Yaskawa INFORM job: X2_38-47,64(1)(90,180)_HARDOX.JBI

/JOB
//NAME X2_38-47,64(1)(90,180)_HARDOX
//POS
///NPOS 504,504,504,30,0,0
///TOOL 0
///POSTYPE PULSE
///PULSE
C00000=-10776,-116726,-133110,1428,79202,268
C00001=-121301,-101656,-130574,-15140,106953,-26685
C00002=-120740,-100574,-124017,-14929,103680,-26084
C00003=-120691,-100743,-123189,-14892,103111,-25997
C00004=-120691,-101012,-123023,-14875,102879,-25968
C00005=-120694,-100727,-123199,-14892,103125,-25999
C00006=-120263,-93974,-120700,-15099,105066,-26103
C00007=-120694,-100727,-123199,-14892,103125,-25999
C00008=-121303,-103883,-129892,-15002,105440,-26491
C00009=-121309,-101301,-130428,-15148,107041,-26699
C00010=-120755,-99767,-124232,-14968,104207,-26155
C00011=-120700,-99774,-123449,-14938,103747,-26079
C00012=-120700,-100712,-122892,-14879,102948,-25979
C00013=-120685,-100384,-123078,-14901,103225,-26009
C00014=-120255,-93653,-120581,-15108,105156,-26112
C00015=-120685,-100384,-123078,-14901,103225,-26009
C00016=-121293,-103472,-129753,-15014,105563,-26504
C00017=-114791,-117911,-130965,-19588,74628,-29967
C00018=-114769,-122713,-124135,-20312,68344,-28880
C00019=-114477,-110584,-116158,-20272,69659,-29005
C00020=-114421,-108517,-114081,-20323,69469,-28951
C00021=-114421,-108669,-113508,-20377,69064,-28879
C00022=-114502,-108614,-114130,-20291,69431,-28974
C00023=-116741,-105993,-113204,-19215,69642,-29832
C00024=-114502,-108614,-114130,-20291,69431,-28974
C00025=-119599,-132627,-121815,-19129,61042,-29452
C00026=-135151,-106131,-113172,-10502,66286,-36044
C00027=-134382,-104032,-112419,-10838,66989,-35834
C00028=-133562,-101757,-111587,-11194,67742,-35614
C00029=-135151,-106131,-113172,-10502,66286,-36044
C00030=-114538,-130880,-126635,-20790,65904,-28347
C00031=-100256,-119338,-132400,-19781,92736,17009
C00032=-115252,-134637,-128783,-15911,82002,19716
C00033=-118597,-124593,-122817,-15129,82811,18454
C00034=-119849,-120977,-120499,-14834,83003,18000
C00035=-119848,-121103,-118880,-14863,81976,18124
C00036=-119849,-120977,-120499,-14834,83003,18000
C00037=-134184,-142802,-124917,-2858,68148,11180
C00038=-133176,-135816,-122960,-3144,70568,11480
C00039=-134184,-142802,-124917,-2858,68148,11180
C00040=-110326,-92448,-108322,-23569,98205,21456
C00041=-112623,-92143,-108201,-23254,97666,20755
C00042=-110326,-92448,-108322,-23569,98205,21456
C00043=-105090,-96290,-113946,-24376,100996,22735
C00044=-105112,-88407,-119445,-25319,107768,21250
C00045=-126458,-130213,-127441,18734,86324,-24062
C00046=-122565,-122494,-122126,18005,86127,-22734
C00047=-121090,-119592,-120022,17718,85999,-22241
C00048=-121089,-119765,-118419,17734,84972,-22390
C00049=-121090,-119592,-120022,17718,85999,-22241
C00050=-121090,-119716,-118696,17731,85160,-22363
C00051=-120619,-113401,-116618,17615,86937,-21943
C00052=-121090,-119716,-118696,17731,85160,-22363
C00053=-120691,-116357,-117549,17638,86049,-22096
C00054=-118089,-117386,-117887,17123,85200,-21315
C00055=-120691,-116357,-117549,17638,86049,-22096
C00056=-125936,-126318,-124843,18636,86589,-23840
C00057=-125953,-122568,-132013,18690,92614,-22924
C00058=-117644,-124381,-130105,-6983,115370,67992
C00059=-119593,-136528,-130318,-6950,109138,67660
C00060=-120425,-140611,-129416,-6959,106433,67520
C00061=-120425,-140322,-128375,-6938,105944,67549
C00062=-120287,-139878,-129033,-6943,106584,67561
C00063=-121808,-147552,-131144,-7070,103828,67181
C00064=-120287,-139878,-129033,-6943,106584,67561
C00065=-117523,-124132,-129146,-6933,114921,68065
C00066=-117634,-108923,-132591,-7489,118176,67765
C00067=-119077,-97405,-129626,-2848,111310,9091
C00068=-112934,-122170,-124968,-9693,82630,11419
C00069=-114889,-112052,-118675,-9157,83718,10686
C00070=-115614,-108714,-115508,-8968,83408,10468
C00071=-115614,-108962,-114752,-8976,82823,10510
C00072=-115614,-108688,-115602,-8966,83479,10463
C00073=-130338,-117040,-117457,5173,77211,4432
C00074=-129550,-114521,-116623,4914,77941,4728
C00075=-131152,-119600,-118288,5441,76463,4123
C00076=-115450,-106601,-114144,-9007,83670,10503
C00077=-117654,-103921,-113183,-8408,84218,9737
C00078=-115450,-106601,-114144,-9007,83670,10503
C00079=-112794,-119726,-122752,-9732,82540,11472
C00080=-112816,-114614,-129461,-9677,89201,10949
C00081=-124267,-125778,-125536,12618,81617,-14637
C00082=-121749,-115664,-119377,11934,82621,-13684
C00083=-120813,-112238,-116231,11692,82317,-13397
C00084=-120812,-112414,-115451,11705,81758,-13450
C00085=-120848,-112349,-116241,11703,82272,-13413
C00086=-119586,-107060,-114409,11339,83657,-12862
C00087=-120848,-112349,-116241,11703,82272,-13413
C00088=-124307,-126037,-124767,12644,81031,-14711
C00089=-124281,-122814,-131176,12539,86499,-14147
C00090=-130647,-155525,-127944,40400,54320,-55258
C00091=-124412,-146323,-123540,36852,53123,-52512
C00092=-122059,-142698,-121760,35413,52755,-51453
C00093=-119008,-142706,-121763,33902,51510,-50382
C00094=-122059,-142698,-121760,35413,52755,-51453
C00095=-119813,-142714,-121776,34308,51836,-50667
C00096=-119829,-137326,-119074,33845,52767,-50322
C00097=-119813,-142714,-121776,34308,51836,-50667
C00098=-119893,-119020,-120433,30427,61542,-47434
C00099=-120958,-113296,-116932,30756,62602,-47571
C00100=-120971,-118070,-117370,31352,60722,-48150
C00101=-120958,-113296,-116932,30756,62602,-47571
C00102=-130647,-155525,-127944,40400,54320,-55258
C00103=-121972,-140000,-127461,3525,22047,-40740
C00104=-114503,-126631,-127045,-28228,88345,-28238
C00105=-115418,-120062,-121213,-28067,87856,-28460
C00106=-115767,-117777,-118144,-28010,87108,-28410
C00107=-115767,-117863,-117333,-28016,86625,-28294
C00108=-115798,-117876,-117463,-28010,86680,-28319
C00109=-115506,-111666,-115391,-28051,88476,-28642
C00110=-115798,-117876,-117463,-28010,86680,-28319
C00111=-114535,-126949,-125608,-28226,87406,-28022
C00112=-81132,-132100,-132064,-22325,96940,-18748
C00113=-82014,-125321,-126186,-22252,96583,-18997
C00114=-82351,-123063,-123074,-22185,95795,-18971
C00115=-82354,-123167,-122323,-22159,95314,-18883
C00116=-82329,-123147,-122467,-22165,95412,-18892
C00117=-83163,-116500,-120334,-22218,97147,-19515
C00118=-82329,-123147,-122467,-22165,95412,-18892
C00119=-81992,-125617,-124767,-22197,95637,-18813
C00120=-81110,-132470,-130662,-22266,95968,-18558
C00121=-88413,-113418,-132573,-32131,117765,-52556
C00122=-88284,-148255,-125485,-32887,110398,-70729
C00123=-90408,-157751,-124889,-32381,105124,-70012
C00124=-91344,-160468,-123864,-32301,103041,-69779
C00125=-91347,-158891,-122215,-32272,102866,-69728
C00126=-106792,-136481,-118062,-29763,111204,-74713
C00127=-106248,-142899,-119829,-29161,109458,-74003
C00128=-106792,-136481,-118062,-29763,111204,-74713
C00129=-72811,-175927,-123443,-35029,98716,-64074
C00130=-76149,-179694,-124176,-35896,96158,-64586
C00131=-72811,-175927,-123443,-35029,98716,-64074
C00132=-69241,-166504,-125806,-34856,105362,-64752
C00133=-100814,-129767,-126176,-13403,120642,-68982
C00134=-124653,-147507,-132240,11278,113041,-68250
C00135=-122082,-159833,-132453,11465,106593,-67927
C00136=-120959,-163108,-131284,11603,104077,-67764
C00137=-120958,-161905,-130051,11594,103939,-67777
C00138=-120958,-161991,-130311,11601,104052,-67766
C00139=-120981,-170969,-132443,11421,100817,-68083
C00140=-120958,-161991,-130311,11601,104052,-67766
C00141=-120973,-170778,-133362,11455,101467,-68019
C00142=-117530,-170630,-133328,12326,101017,-66845
C00143=-120973,-170778,-133362,11455,101467,-68019
C00144=-124784,-154865,-133680,10989,110216,-68576
C00145=-122322,-137878,-131274,-5971,121779,-67906
C00146=-120548,-145044,-127252,-18536,119036,-66813
C00147=-120555,-156847,-127343,-17506,113306,-65855
C00148=-120558,-160498,-126573,-17182,111059,-65507
C00149=-120558,-158961,-124938,-17154,110851,-65476
C00150=-120618,-159187,-125406,-17199,111003,-65522
C00151=-120626,-166810,-127194,-16864,108302,-65121
C00152=-120618,-159187,-125406,-17199,111003,-65522
C00153=-120603,-144021,-125705,-18473,118618,-66761
C00154=-115387,-132374,-123926,-32562,106734,-81694
C00155=-118372,-141379,-123449,-32107,101406,-81342
C00156=-119656,-144207,-122551,-32012,99204,-81226
C00157=-119656,-143343,-121080,-31963,98811,-81114
C00158=-119656,-144508,-123075,-32029,99348,-81268
C00159=-131320,-114613,-113969,-28597,111497,-86004
C00160=-131699,-120616,-115930,-28265,109708,-85685
C00161=-131320,-114613,-113969,-28597,111497,-86004
C00162=-105239,-169544,-124716,-37289,88926,-74807
C00163=-108884,-170779,-124983,-37802,86985,-75650
C00164=-105239,-169544,-124716,-37289,88926,-74807
C00165=-99694,-161827,-127351,-36723,95805,-74832
C00166=-131992,-100814,-126478,-21663,116809,46067
C00167=-134007,-144842,-130967,-18968,105768,42043
C00168=-134012,-143545,-127522,-18820,104388,42265
C00169=-134287,-143929,-127856,-18860,104334,42172
C00170=-133739,-135079,-123901,-19000,106464,42030
C00171=-134287,-143184,-126185,-18799,103720,42271
C00172=-134064,-144330,-127677,-2767,111202,58459
C00173=-134007,-143438,-127424,-2760,111507,58474
C00174=-135126,-137550,-119428,14300,119099,83463
C00175=-134030,-140788,-121209,15013,118595,84384
C00176=-134030,-142235,-124150,15187,119626,84533
C00177=-119630,-122416,-133334,16028,118546,61096
C00178=-134341,-125466,-134740,10815,104436,21672
C00179=-120614,-100166,-121253,7350,89365,-11707
C00180=-120622,-93660,-109595,7359,85566,-11930
C00181=-122164,-90812,-108950,7802,86761,-12352
C00182=-122198,-95853,-109304,7828,84412,-12509
C00183=-122164,-91688,-107664,7808,85529,-12428
C00184=-120622,-94101,-108793,7365,84850,-11972
C00185=-122951,-73862,-99576,-7929,88190,4985
C00186=-120621,-96600,-101892,-16342,67221,11741
C00187=-120621,-96191,-103793,-16192,68548,11553
C00188=-120639,-92247,-111396,-15618,75005,10677
C00189=-188010,-107595,-125638,17104,94805,-24250
C00190=-188020,-110122,-123495,17031,92300,-24603
C00191=-187252,-116827,-124472,16830,89421,-24740
C00192=-188438,-109992,-122083,17102,91614,-24840
C00193=-188123,-110345,-123595,17051,92269,-24642
C00194=-188114,-107825,-125741,17124,94773,-24289
C00195=-177438,-122732,-133224,14695,89877,-21402
C00196=-133569,-113989,-134534,14289,94663,-20149
C00197=-119624,-110386,-135117,7911,77851,-79525
C00198=-120615,-106635,-127104,8473,74968,-80030
C00199=-127138,-106639,-125023,15586,75013,-81251
C00200=-130661,-111022,-125418,19776,73192,-82197
C00201=-120615,-106612,-127117,8473,74988,-80029
C00202=-122620,-125184,-116655,35316,53565,-49443
C00203=-120598,-121294,-114839,33833,53482,-48472
C00204=-120551,-127900,-115071,35213,50759,-49502
C00205=-120377,-147941,-114075,41532,42004,-53628
C00206=-120733,-119186,-113678,30224,65857,-57863
C00207=-122683,-120749,-115245,30946,66698,-58435
C00208=-127694,-124296,-119025,32687,68997,-59841
C00209=-127721,-118762,-131765,31151,78153,-27047
C00210=-126237,-112945,-130032,468,65797,-4909
C00211=-102361,-117345,-122757,-6013,83638,2551
C00212=-102141,-118134,-119975,-6094,81548,2725
C00213=-99061,-100059,-114136,-7526,92006,6303
C00214=-118448,-105217,-116092,-2994,89929,-3052
C00215=-122253,-105715,-115580,-4099,87909,4316
C00216=-120609,-124185,-121101,-4570,77097,5239
C00217=-120610,-123821,-123927,-4542,79018,5168
C00218=-108948,-109237,-131335,-7817,91844,8301
C00219=-115305,-101104,-129841,-7326,117578,44729
C00220=-120606,-132359,-125648,-5649,119733,79611
C00221=-120606,-131978,-122596,-5547,118059,79698
C00222=-120699,-131888,-121364,-5538,117345,79699
C00223=-120606,-132064,-121373,-5500,117266,79739
C00224=-120606,-131696,-121291,-5509,117403,79735
C00225=-120606,-131546,-119742,-13806,116783,67512
C00226=-120606,-131851,-120987,-13891,117375,67436
C00227=-120606,-132395,-123921,-14113,118858,67242
C00228=-111305,-120759,-132293,-17375,98141,32748
C00229=-120609,-124691,-119154,-16638,71592,14867
C00230=-120609,-124440,-116582,-16774,70197,15066
C00231=-120609,-124277,-115533,-16830,69659,15144
C00232=-120609,-125082,-119997,8806,76841,-5950
C00233=-120609,-124819,-119897,8803,76914,-5945
C00234=-120609,-124768,-117835,18246,76542,-19045
C00235=-120609,-124884,-118955,18205,77141,-18954
C00236=-120609,-124961,-121688,18108,78705,-18718
C00237=-132640,-106780,-128323,23054,110263,28369
C00238=-120602,-139315,-124713,24306,112781,84362
C00239=-120602,-138068,-121544,24057,111582,84094
C00240=-120602,-137520,-120260,23964,111115,83992
C00241=-111171,-137450,-123178,3338,116163,79197
C00242=-120602,-139000,-123563,90,115805,75571
C00243=-109330,-134151,-116420,-27663,112170,68648
C00244=-107669,-134044,-117364,-27346,113285,69054
C00245=-103576,-133216,-119553,-26575,116197,70036
C00246=-103610,-135048,-130246,-28186,121222,68648
C00247=-111190,-129681,-128447,-36946,96833,72948
C00248=-111854,-129032,-128166,-43025,93670,81713
C00249=-147502,-118658,-119533,-35927,77679,72524
C00250=-147511,-119004,-116560,-36172,76036,73070
C00251=-147515,-119022,-115332,-36276,75411,73279
C00252=-147547,-116234,-125968,-15022,114340,70681
C00253=-147515,-116012,-125840,-15022,114380,70688
C00254=-147502,-115929,-125780,-17177,108602,60467
C00255=-147494,-115895,-125723,-16722,102508,50684
C00256=-147493,-115916,-125679,-13964,96968,41110
C00257=-147497,-115970,-125656,-10645,93613,33926
C00258=-147501,-116025,-125648,-8199,92025,29507
C00259=-147506,-116072,-125646,-5516,90867,25066
C00260=-147508,-116095,-125646,-5516,90856,25066
C00261=-147505,-115163,-126691,-5523,91973,25018
C00262=-147498,-112805,-128627,-5545,94366,24915
C00263=-120610,-124729,-127429,5691,77135,-5542
C00264=-120610,-125478,-124917,5733,75213,-5631
C00265=-121145,-125062,-125115,1467,77680,-1578
C00266=-93224,-108496,-118221,-17160,84932,17314
C00267=-100404,-109639,-120638,-9099,85725,5885
C00268=-100577,-112155,-122052,-6607,85486,-528
C00269=-115338,-131033,-127093,4056,76541,-4536
C00270=-121145,-125062,-125115,1467,77680,-1578
C00271=-113474,-126239,-125199,-4571,76718,-3065
C00272=-116327,-126679,-125338,-2161,76267,-5597
C00273=-113490,-126055,-125151,-4559,76778,-3077
C00274=-117667,-122970,-124192,-3214,77575,-4511
C00275=-120712,-121109,-123606,-2232,78069,-5542
C00276=-125774,-129632,-127388,3161,76112,-11172
C00277=-120611,-124694,-128184,1477,78993,-9385
C00278=2000,-120083,-131752,1890,40973,0
C00279=-15972,-110889,-128286,-10965,59905,-43045
C00280=-101389,-60822,-75148,6919,68546,-70102
C00281=-115790,69230,64798,-8053,66131,-71909
C00282=-120830,71540,61874,-4756,55589,-66514
C00283=-120535,76858,72419,-5134,51864,-66212
C00284=-120418,79487,77321,-5314,50212,-66075
C00285=-120418,81305,81326,-5435,48689,-65991
C00286=-120418,79487,77321,-5314,50212,-66075
C00287=-121101,73566,71896,-4942,50464,-66384
C00288=-120640,77942,77238,-5256,49458,-66131
C00289=-121101,73566,71896,-4942,50464,-66384
C00290=-121527,66226,57370,-4418,55590,-66797
C00291=-120817,46858,51705,6808,46216,-80289
C00292=-120487,52530,62238,7041,42645,-80409
C00293=-120357,55197,66992,7170,41090,-80474
C00294=-120357,57219,71131,7393,39594,-80606
C00295=-120357,55197,66992,7170,41090,-80474
C00296=-121171,51687,64922,7778,40638,-80922
C00297=-120657,55397,69123,7546,39918,-80729
C00298=-121171,51687,64922,7778,40638,-80922
C00299=-121648,43436,49847,7373,45678,-80715
C00300=-109578,66950,51259,-9202,73878,-70224
C00301=-101389,-60822,-75148,6919,68546,-70102
C00302=-96929,-90691,-89138,5080,61517,-23019
C00303=-96929,-90691,-89138,5080,61517,27168
C00304=-133997,38575,-5386,4879,105902,64390
C00305=-134430,35731,-4221,4855,103756,64161
C00306=-134605,34491,-3252,4839,102536,64054
C00307=-134604,34193,-2477,4825,101908,64030
C00308=-134605,34666,-3678,4847,102887,64068
C00309=-133324,38381,1851,4717,101326,64430
C00310=-133984,36157,-436,4773,101627,64224
C00311=-133324,38381,1851,4717,101326,64430
C00312=-132740,42105,45,4739,104308,64739
C00313=-134038,40743,-3018,12196,109842,66951
C00314=-134155,37294,-2552,12029,107844,66703
C00315=-134138,36860,-901,11936,106627,66584
C00316=-134138,36533,-42,11887,105945,66515
C00317=-134138,36618,-275,11900,106128,66533
C00318=-134308,36004,-906,11910,106222,66482
C00319=-134138,36772,-681,11923,106449,66566
C00320=-133552,41863,-495,12102,108819,67011
C00321=-143157,-5596,-33734,3459,84138,-17748
C00322=-146617,-6443,-23161,4534,77380,-19112
C00323=-149281,-2495,-17370,9500,77350,-25048
C00324=-149281,-2461,-16373,9521,76762,-25094
C00325=-149281,-2503,-17669,9494,77528,-25035
C00326=-148457,-726,-16200,9269,77441,-24757
C00327=-149281,-2503,-17669,9494,77528,-25035
C00328=-157589,4412,-9593,22718,80450,-41052
C00329=-157226,5016,-8132,22675,79802,-41042
C00330=-156592,4240,-8798,22542,79640,-40841
C00331=-157226,4947,-9136,22642,80340,-40940
C00332=-149281,-2387,-22338,9412,80423,-24814
C00333=-159526,23962,790,32225,80504,55500
C00334=-158922,24925,5721,32299,78113,55050
C00335=-158153,25889,7618,32183,77247,55110
C00336=-158153,25992,9261,32290,76429,54873
C00337=-158153,25975,9034,32275,76541,54905
C00338=-159336,23803,6937,32538,77140,54603
C00339=-159336,23824,7234,32557,76994,54560
C00340=-158542,24868,8237,32379,76622,54771
C00341=-158626,24722,8098,32398,76663,54749
C00342=-158626,24746,8414,32418,76509,54705
C00343=-158626,24723,8130,32399,76648,54745
C00344=-159596,23128,6599,32614,77122,54493
C00345=-159596,23153,6932,32637,76960,54446
C00346=-159062,24432,8187,32525,76656,54571
C00347=-159244,23446,6313,32496,77274,54679
C00348=-160967,21427,101,32642,80299,54873
C00349=-147551,27169,-6215,28445,81493,60312
C00350=-147017,27605,-1759,28452,79091,59917
C00351=-146493,28433,829,28390,77886,59816
C00352=-146493,28355,1445,28429,77515,59723
C00353=-146493,28387,1187,28413,77670,59762
C00354=-147642,25561,-1571,28744,78267,59478
C00355=-147642,25516,-1231,28765,78061,59427
C00356=-146933,27046,255,28560,77712,59607
C00357=-147010,26749,-33,28581,77761,59589
C00358=-147010,26722,196,28596,77625,59555
C00359=-147010,26770,-196,28572,77860,59614
C00360=-147964,24407,-2486,28847,78350,59377
C00361=-147964,24325,-1833,28887,77960,59278
C00362=-147292,26053,-161,28694,77611,59445
C00363=-147523,24411,-2449,28713,78186,59502
C00364=-149162,23542,-7999,28991,81344,59682
C00365=-148025,26294,-7040,28591,81698,60189
C00366=-147485,26714,-2602,28593,79299,59793
C00367=-147271,26975,-740,28610,78335,59633
C00368=-147270,26798,747,28702,77445,59410
C00369=-147271,26975,-740,28610,78335,59633
C00370=-147888,25428,-868,28863,77908,59292
C00371=-147063,27300,949,28626,77494,59501
C00372=-147888,25428,-868,28863,77908,59292
C00373=-148652,24637,-7261,28828,81272,59852
C00374=-129846,-17397,-52274,16165,101048,68229
C00375=-103949,-6271,-30701,7884,96105,76175
C00376=-94102,16895,-5866,4380,94047,79161
C00377=-94024,14878,-3719,4358,91692,79105
C00378=-93993,14152,-2780,4351,90742,79083
C00379=-93993,14213,-1554,4335,90021,79057
C00380=-93993,14202,-1750,4335,90136,79060
C00381=-93544,18458,2169,4295,89888,79203
C00382=-93544,18476,2442,4295,89728,79198
C00383=-93713,17041,1146,4310,89799,79144
C00384=-93671,17336,1418,4307,89780,79158
C00385=-93671,17356,1712,4307,89607,79151
C00386=-93671,17342,1501,4307,89730,79155
C00387=-93486,20302,4269,4303,89540,79209
C00388=-93873,20584,4779,4336,89392,79073
C00389=-94001,18334,2673,4347,89541,79036
C00390=-94106,19042,2519,4357,90004,79017
C00391=-93796,22544,1176,4343,92603,79213
C00392=-95224,-25687,-42365,27028,60157,72238
C00393=-94111,-23276,-36997,26973,57954,72128
C00394=-93597,-19509,-33603,26734,57655,72271
C00395=-93597,-19504,-31914,27029,56727,72023
C00396=-93597,-19510,-32243,26972,56905,72072
C00397=-93990,-24549,-35870,27293,56712,71846
C00398=-93990,-24538,-35459,27369,56492,71783
C00399=-93788,-21252,-33109,27186,56644,71914
C00400=-93840,-21553,-33328,27220,56642,71889
C00401=-93840,-21543,-33005,27278,56468,71842
C00402=-93840,-21553,-33351,27216,56655,71894
C00403=-94357,-24968,-35787,27577,56595,71647
C00404=-94357,-24947,-35259,27673,56314,71569
C00405=-94013,-22711,-33670,27433,56354,71733
C00406=-93814,-23881,-35617,27147,56823,71950
C00407=-98687,-54699,-75805,10421,73482,70446
C00408=-149776,12587,-27486,12781,89603,-18869
C00409=-147726,21450,-15619,10072,89467,-18633
C00410=-146190,28089,-6729,8043,89366,-18457
C00411=-138712,21584,-10452,-6744,81967,66
C00412=-138085,14099,-20532,-6917,84360,139
C00413=-145864,23955,-12684,8284,88428,-27874
C00414=-146885,25936,-8147,8552,86771,-28313
C00415=-147056,24986,-14909,8600,90423,-28118
C00416=-133623,24371,-15503,-12505,92341,-3955
C00417=-141603,20096,-23343,17631,90771,45924
C00418=-175362,59573,37827,46975,74531,48445
C00419=-174398,62305,44598,47324,72110,47721
C00420=-174059,64572,48196,47497,71206,47437
C00421=-174678,72270,57247,48014,70425,46715
C00422=-172628,50226,32658,43982,63214,47275
C00423=-173442,46522,25111,43389,65629,48000
C00424=-175751,57855,36014,51960,82937,49775
C00425=-174440,56084,37605,51944,81006,49370
C00426=-173757,55485,37843,51901,80337,49352
C00427=-174241,61252,44330,52087,79962,48874
C00428=-175386,74687,58791,55260,88042,49507
C00429=-176596,75085,57687,55306,89275,49600
C00430=-162891,39596,10758,46944,80889,54952
C00431=-161747,40468,15313,46928,78664,54425
C00432=-163273,53880,32001,50799,82657,52192
C00433=-162010,46460,23909,50499,82720,52878
C00434=-160571,34350,9025,46543,78569,54946
C00435=-161741,33529,4546,46578,80799,55455
C00436=-147996,42947,122,12460,106294,61459
C00437=-148226,40262,1426,12324,104193,61162
C00438=-146766,53866,17608,9771,108156,61626
C00439=-145306,48527,11741,9899,108797,62196
C00440=-146773,35404,-3590,12275,104564,61692
C00441=-146547,41093,-8751,12742,110494,62402
C00442=-170472,-48867,-31078,12436,82300,51309
C00443=-161833,-30139,-32162,12294,91042,55174
C00444=-111128,62365,52281,-11955,55160,-64549
C00445=-111043,67239,62048,-12539,51743,-64100
C00446=-108427,49473,54066,-27881,35011,-61543
C00447=-110512,52951,57928,-26501,33808,-62418
C00448=-113115,71610,67239,-11613,50506,-64854
C00449=-113215,66301,56846,-11015,54091,-65302
C00450=-121898,77388,65564,1855,57299,-70150
C00451=-121470,82378,75801,1732,53556,-70040
C00452=-123195,67922,64647,6849,45018,-71451
C00453=-122125,64607,60584,6056,45727,-70899
C00454=-120225,78262,70725,1119,54542,-69513
C00455=-120651,73746,61164,1269,58111,-69644
C00456=-113189,52303,49996,7645,51731,-77534
C00457=-112734,56976,59397,7777,48333,-77603
C00458=-114820,45850,55114,15931,36430,-80431
C00459=-110545,39461,48380,12117,36535,-77984
C00460=-108220,49577,51136,5183,49245,-75539
C00461=-108655,45336,42401,5185,52457,-75559
C00462=-161833,-30139,-32162,12294,91042,55174
C00463=-170472,-47446,-27408,12476,80805,51159
C00464=-92809,-22406,-39596,-2559,87564,76845
C00465=-93205,-23584,-36354,-2491,84954,76766
C00466=-93256,-22757,-34134,-2485,84011,76766
C00467=-94635,-22284,-33796,-2233,84005,76304
C00468=-94250,-23197,-36080,-2300,84954,76417
C00469=-93848,-22027,-39325,-2370,87561,76502
C00470=-94651,-21766,-39138,7100,89212,77956
C00471=-94455,-23170,-36061,7070,86599,77874
C00472=-94691,-22224,-33752,7109,85688,77745
C00473=-93741,-22621,-34036,6956,85577,78058
C00474=-93466,-23543,-36325,6911,86486,78200
C00475=-93670,-22147,-39411,6941,89101,78276
C00476=-92980,-26767,-42567,6357,64758,77223
C00477=-92830,-24983,-37315,6405,62444,77148
C00478=-93074,-23230,-34736,6569,61782,77018
C00479=-94403,-22562,-34257,7239,61942,76525
C00480=-95090,-24132,-36711,8569,62895,76288
C00481=-95328,-25868,-41938,8524,65219,76375
C00482=-95261,-25907,-41974,7480,65026,76408
C00483=-95085,-24145,-36729,7536,62706,76321
C00484=-95077,-22533,-34315,7574,62052,76278
C00485=-94015,-22863,-34552,7040,61932,76670
C00486=-92783,-25001,-37319,5340,62272,77201
C00487=-92870,-26808,-42587,5281,64581,77276
C00488=-120452,-88146,-86102,21652,66713,67139
C00489=-165262,-16782,-33522,47685,80918,53825
C00490=-161018,-5245,-12472,47809,73866,52405
C00491=-160379,-4160,-10611,47798,73123,52356
C00492=-157904,-13140,-17700,47336,71641,52867
C00493=-158239,-15440,-20419,47297,72158,52954
C00494=-159752,-17175,-25374,47188,74446,53337
C00495=-148723,45367,2700,12479,106062,61188
C00496=-148955,42713,4001,12346,103979,60892
C00497=-149715,44338,7129,12324,103024,60537
C00498=-146495,33091,-4314,12210,103798,61708
C00499=-146015,32884,-6147,12245,104729,61965
C00500=-145791,35660,-7470,12388,106889,62265
C00501=-109011,-26713,-50438,8452,98222,74634
C00502=-84134,-123556,-96733,5664,74963,81774
C00503=-10907,-117335,-90652,-18762,63715,-59495
BC00000=165820,667836,1075229
BC00001=35816,1008911,1075175
BC00002=35816,1008911,1075175
BC00003=35816,1008911,1075175
BC00004=35816,1008911,1075175
BC00005=35816,1008911,1075175
BC00006=35816,1008911,1075175
BC00007=35816,1008911,1075175
BC00008=35816,1008911,1075175
BC00009=81778,1000994,1075175
BC00010=81778,1000994,1075175
BC00011=81778,1000994,1075175
BC00012=81778,1000994,1075175
BC00013=81778,1000994,1075175
BC00014=81778,1000994,1075175
BC00015=81778,1000994,1075175
BC00016=81778,1000994,1075175
BC00017=183238,908205,1075175
BC00018=183238,908205,1075175
BC00019=183238,908205,1075175
BC00020=183238,908205,1075175
BC00021=183238,908205,1075175
BC00022=183238,908205,1075175
BC00023=183238,908205,1075175
BC00024=183238,908205,1075175
BC00025=183238,908205,1075175
BC00026=183238,908205,1075175
BC00027=183238,908205,1075175
BC00028=183238,908205,1075175
BC00029=183238,908205,1075175
BC00030=183238,908205,1075175
BC00031=277080,941460,1075175
BC00032=289789,946711,1075175
BC00033=289789,946711,1075175
BC00034=289789,946711,1075175
BC00035=289789,946711,1075175
BC00036=289789,946711,1075175
BC00037=289789,946711,1075175
BC00038=289789,946711,1075175
BC00039=289789,946711,1075175
BC00040=289789,946711,1075175
BC00041=289789,946711,1075175
BC00042=289789,946711,1075175
BC00043=289789,946711,1075175
BC00044=289789,946711,1075175
BC00045=261300,945494,1075175
BC00046=261300,945494,1075175
BC00047=261300,945494,1075175
BC00048=261300,945494,1075175
BC00049=261300,945494,1075175
BC00050=261300,945494,1075175
BC00051=261300,945494,1075175
BC00052=261300,945494,1075175
BC00053=261300,945494,1075175
BC00054=261300,945494,1075175
BC00055=261300,945494,1075175
BC00056=261300,945494,1075175
BC00057=261300,945494,1075175
BC00058=293747,972847,1075175
BC00059=293747,972847,1075175
BC00060=293747,972847,1075175
BC00061=293747,972847,1075175
BC00062=293747,972847,1075175
BC00063=293747,972847,1075175
BC00064=293747,972847,1075175
BC00065=293747,972847,1075175
BC00066=293747,958005,1075175
BC00067=262329,883284,1075175
BC00068=265687,860722,1075175
BC00069=265687,860722,1075175
BC00070=265687,860722,1075175
BC00071=265687,860722,1075175
BC00072=265687,860722,1075175
BC00073=265687,860722,1075175
BC00074=265687,860722,1075175
BC00075=265687,860722,1075175
BC00076=265687,860722,1075175
BC00077=265687,860722,1075175
BC00078=265687,860722,1075175
BC00079=265687,860722,1075175
BC00080=265687,860722,1075175
BC00081=272052,840663,1075175
BC00082=272052,840663,1075175
BC00083=272052,840663,1075175
BC00084=272052,840663,1075175
BC00085=272052,840663,1075175
BC00086=272052,840663,1075175
BC00087=272052,840663,1075175
BC00088=272052,840663,1075175
BC00089=272052,840663,1075175
BC00090=294078,933568,1075175
BC00091=294078,933568,1075175
BC00092=294078,933568,1075175
BC00093=294078,933568,1075175
BC00094=294078,933568,1075175
BC00095=294078,933568,1075175
BC00096=294078,933568,1075175
BC00097=294078,933568,1075175
BC00098=294078,933568,1075175
BC00099=294078,933568,1075175
BC00100=294078,933568,1075175
BC00101=294078,933568,1075175
BC00102=294078,933568,1075175
BC00103=350010,851645,1075175
BC00104=398174,950083,1075175
BC00105=398174,950083,1075175
BC00106=398174,950083,1075175
BC00107=398174,950083,1075175
BC00108=398174,950083,1075175
BC00109=398174,950083,1075175
BC00110=398174,950083,1075175
BC00111=398174,950083,1075175
BC00112=398174,954074,1075175
BC00113=398174,954074,1075175
BC00114=398174,954074,1075175
BC00115=398174,954074,1075175
BC00116=398174,954074,1075175
BC00117=398174,954074,1075175
BC00118=398174,954074,1075175
BC00119=398174,954074,1075175
BC00120=398174,954074,1075175
BC00121=398174,870681,1075175
BC00122=398174,817728,1075175
BC00123=398174,817728,1075175
BC00124=398174,817728,1075175
BC00125=398174,817728,1075175
BC00126=398174,817728,1075175
BC00127=398174,817728,1075175
BC00128=398174,817728,1075175
BC00129=398174,817728,1075175
BC00130=398174,817728,1075175
BC00131=398174,817728,1075175
BC00132=398174,817728,1075175
BC00133=396448,827169,1075175
BC00134=394822,829620,1075175
BC00135=394822,829620,1075175
BC00136=394822,829620,1075175
BC00137=394822,829620,1075175
BC00138=394822,829620,1075175
BC00139=394822,829620,1075175
BC00140=394822,829620,1075175
BC00141=394822,829620,1075175
BC00142=394822,829620,1075175
BC00143=394822,829620,1075175
BC00144=394822,829620,1075175
BC00145=355383,833896,1075175
BC00146=324600,845042,1075175
BC00147=324600,845042,1075175
BC00148=324600,845042,1075175
BC00149=324600,845042,1075175
BC00150=324600,845042,1075175
BC00151=324600,845042,1075175
BC00152=324600,845042,1075175
BC00153=324600,845042,1075175
BC00154=311941,807883,1075175
BC00155=311941,807883,1075175
BC00156=311941,807883,1075175
BC00157=311941,807883,1075175
BC00158=311941,807883,1075175
BC00159=311941,807883,1075175
BC00160=311941,807883,1075175
BC00161=311941,807883,1075175
BC00162=311941,807883,1075175
BC00163=311941,807883,1075175
BC00164=311941,807883,1075175
BC00165=311941,807883,1075175
BC00166=316281,962914,1075175
BC00167=312573,990264,1075175
BC00168=307903,987774,1075175
BC00169=306034,986778,1075175
BC00170=306034,986778,1075175
BC00171=306034,986778,1075175
BC00172=283260,992694,1075175
BC00173=316930,973741,1075175
BC00174=283185,985095,1075172
BC00175=281644,987513,1075175
BC00176=279107,993102,1075175
BC00177=280151,960541,1075175
BC00178=281317,877250,1075175
BC00179=282638,819792,1075175
BC00180=284858,824834,1075175
BC00181=285747,826851,1075175
BC00182=285747,826851,1075175
BC00183=285747,826851,1075175
BC00184=239186,852971,1075175
BC00185=275413,838907,1075175
BC00186=285600,832969,1075175
BC00187=288466,826898,1075175
BC00188=288466,826898,1075175
BC00189=136054,1003977,1075175
BC00190=136349,1009357,1075175
BC00191=136467,1011509,1075175
BC00192=85590,1020321,1075175
BC00193=85472,1018169,1075175
BC00194=85177,1012789,1075175
BC00195=85177,867663,1075175
BC00196=394575,855601,1075175
BC00197=335365,938803,1075175
BC00198=336708,934958,1075175
BC00199=337245,935767,1075175
BC00200=337268,942708,1075175
BC00201=336730,941898,1075175
BC00202=295940,927161,1075175
BC00203=295940,927161,1075175
BC00204=295940,927161,1075175
BC00205=295940,927161,1075175
BC00206=295940,927161,1075175
BC00207=295940,927161,1075175
BC00208=295940,927161,1075175
BC00209=295940,927161,1075175
BC00210=393681,912027,1075175
BC00211=398174,921728,1075175
BC00212=398174,926962,1075175
BC00213=398174,928620,1075175
BC00214=364761,938622,1075175
BC00215=369199,937365,1075175
BC00216=369642,935240,1075175
BC00217=370750,929927,1075175
BC00218=370750,848394,1075175
BC00219=340693,834439,1075175
BC00220=313140,829466,1075175
BC00221=312428,824087,1075175
BC00222=312144,821935,1075175
BC00223=307365,821950,1075175
BC00224=268115,822068,1075172
BC00225=280175,821657,1075175
BC00226=281271,823684,1075175
BC00227=284011,828752,1075175
BC00228=290728,897938,1075175
BC00229=293762,929183,1075175
BC00230=290448,934424,1075175
BC00231=289122,936520,1075175
BC00232=241729,942952,1075175
BC00233=279832,936352,1075175
BC00234=264136,939681,1075175
BC00235=262547,937931,1075175
BC00236=258574,933557,1075175
BC00237=314949,872913,1075175
BC00238=378471,827894,1075175
BC00239=380915,822749,1075175
BC00240=381893,820691,1075175
BC00241=398174,825891,1075175
BC00242=361449,826034,1075175
BC00243=398174,815367,1075175
BC00244=398174,817132,1075175
BC00245=398174,821543,1075175
BC00246=398174,821543,1075175
BC00247=256492,965748,1075175
BC00248=237924,1001427,1075175
BC00249=237924,1015453,1075175
BC00250=232933,1013664,1075175
BC00251=230937,1012949,1075175
BC00252=178459,1050835,1075175
BC00253=213013,1031453,1075175
BC00254=227041,1020134,1075175
BC00255=235513,1004484,1075175
BC00256=237128,986927,1075175
BC00257=233266,973358,1075175
BC00258=228054,964181,1075175
BC00259=223178,957936,1075175
BC00260=220682,955545,1075175
BC00261=222343,954677,1075175
BC00262=225664,952941,1075175
BC00263=141848,914666,1075175
BC00264=143128,920299,1075175
BC00265=148671,926943,1075175
BC00266=143639,922553,1075175
BC00267=137651,924704,1075175
BC00268=129694,927561,1075175
BC00269=134120,930846,1075175
BC00270=148671,926943,1075175
BC00271=116938,942468,1075175
BC00272=115693,943064,1075175
BC00273=111414,945116,1075175
BC00274=111414,945116,1075175
BC00275=111414,945116,1075175
BC00276=110923,942951,1075175
BC00277=109940,938621,1075175
BC00278=131749,675704,1075175
BC00279=21214,672831,429902
BC00280=66815,724118,419761
BC00281=110240,772957,337669
BC00282=136729,789553,283981
BC00283=136729,789553,283981
BC00284=136729,789553,283981
BC00285=136729,789553,283981
BC00286=136729,789553,283981
BC00287=136729,789553,283981
BC00288=136729,789553,283981
BC00289=136729,789553,283981
BC00290=136729,789553,283981
BC00291=163194,789553,386705
BC00292=163194,789553,386705
BC00293=163194,789553,386705
BC00294=163194,789553,386705
BC00295=163194,789553,386705
BC00296=163194,789553,386705
BC00297=163194,789553,386705
BC00298=163194,789553,386705
BC00299=163194,789553,386705
BC00300=110240,772957,337669
BC00301=66815,724118,419761
BC00302=66815,670858,419761
BC00303=252765,670858,277331
BC00304=322808,760288,131711
BC00305=322808,760288,131711
BC00306=322808,760288,131711
BC00307=322808,760288,131711
BC00308=322808,760288,131711
BC00309=322808,760288,131711
BC00310=322808,760288,131711
BC00311=322808,760288,131711
BC00312=322808,760288,131711
BC00313=340407,752653,125690
BC00314=340407,752653,125690
BC00315=340407,752653,125690
BC00316=340407,752653,125690
BC00317=340407,752653,125690
BC00318=340407,752653,125690
BC00319=340407,752653,125690
BC00320=340407,752653,125690
BC00321=309477,783812,200910
BC00322=309477,783812,200910
BC00323=309477,783812,200910
BC00324=309477,783812,200910
BC00325=309477,783812,200910
BC00326=309477,783812,200910
BC00327=309477,783812,200910
BC00328=309477,783812,200910
BC00329=309477,783812,200910
BC00330=309477,783812,200910
BC00331=309477,783812,200910
BC00332=309477,783812,200910
BC00333=335534,789553,204922
BC00334=335534,789553,204922
BC00335=335534,789553,204922
BC00336=335534,789553,204922
BC00337=335534,789553,204922
BC00338=335534,789553,204922
BC00339=335534,789553,204922
BC00340=335534,789553,204922
BC00341=335534,789553,204922
BC00342=335534,789553,204922
BC00343=335534,789553,204922
BC00344=335534,789553,204922
BC00345=335534,789553,204922
BC00346=335534,789553,204922
BC00347=335534,789553,204922
BC00348=335534,789553,204922
BC00349=344006,752651,139062
BC00350=344006,752651,139062
BC00351=344005,752652,139060
BC00352=344005,752652,139060
BC00353=344005,752652,139060
BC00354=344005,752652,139060
BC00355=344005,752652,139060
BC00356=344005,752652,139060
BC00357=344005,752652,139060
BC00358=344005,752652,139060
BC00359=344005,752652,139060
BC00360=344005,752652,139060
BC00361=344005,752652,139060
BC00362=344005,752652,139060
BC00363=344005,752652,139060
BC00364=344006,752651,139062
BC00365=374489,733638,136084
BC00366=374489,733638,136084
BC00367=374489,733638,136084
BC00368=374489,733638,136084
BC00369=374489,733638,136084
BC00370=374489,733638,136084
BC00371=374489,733638,136084
BC00372=374489,733638,136084
BC00373=374489,733638,136084
BC00374=300933,750795,218908
BC00375=283893,750061,250495
BC00376=276320,749735,264534
BC00377=276320,749735,264534
BC00378=276320,749735,264534
BC00379=276320,749735,264532
BC00380=276320,749735,264532
BC00381=276320,749735,264532
BC00382=276320,749735,264532
BC00383=276320,749735,264532
BC00384=276320,749735,264532
BC00385=276320,749735,264532
BC00386=276320,749735,264532
BC00387=276320,749736,264531
BC00388=276320,749736,264531
BC00389=276320,749736,264531
BC00390=276320,749736,264531
BC00391=276320,749735,264534
BC00392=248857,763770,138691
BC00393=248857,763770,138691
BC00394=248857,763770,138691
BC00395=248857,763770,138691
BC00396=248857,763770,138691
BC00397=248857,763770,138691
BC00398=248857,763770,138691
BC00399=248857,763770,138691
BC00400=248857,763770,138691
BC00401=248857,763770,138691
BC00402=248857,763770,138691
BC00403=248857,763770,138691
BC00404=248857,763770,138691
BC00405=248857,763770,138691
BC00406=248857,763770,138691
BC00407=248857,763770,138691
BC00408=315051,758770,94341
BC00409=315051,758770,94341
BC00410=315051,758770,94341
BC00411=315051,758770,94341
BC00412=315051,758770,94341
BC00413=315051,758770,94341
BC00414=315051,758770,94341
BC00415=315051,758770,94341
BC00416=315051,758770,94341
BC00417=315051,758770,94341
BC00418=398174,761952,129173
BC00419=398174,761952,129173
BC00420=398174,761952,129173
BC00421=398174,761952,129173
BC00422=398174,761952,129173
BC00423=398174,761952,129173
BC00424=366295,778309,120132
BC00425=366295,778309,120132
BC00426=366295,778309,120132
BC00427=366295,778309,120132
BC00428=366295,778309,120132
BC00429=366295,778309,120132
BC00430=398174,729290,94227
BC00431=398174,729290,94227
BC00432=398174,729290,94227
BC00433=398174,729290,94227
BC00434=398174,729290,94227
BC00435=398174,729290,94227
BC00436=382568,752165,121199
BC00437=382568,752165,121199
BC00438=382568,752165,121199
BC00439=382568,752165,121199
BC00440=382568,752165,121199
BC00441=382568,752165,121199
BC00442=382568,668969,422236
BC00443=167343,668969,639457
BC00444=112241,789553,268043
BC00445=112241,789553,268043
BC00446=112241,789553,268043
BC00447=112241,789553,268043
BC00448=112241,789553,268043
BC00449=112241,789553,268043
BC00450=121114,789553,252467
BC00451=121114,789553,252467
BC00452=121114,789553,252467
BC00453=121114,789553,252467
BC00454=121114,789553,252467
BC00455=121114,789553,252467
BC00456=121337,789553,329708
BC00457=121337,789553,329708
BC00458=121337,789553,329708
BC00459=121337,789553,329708
BC00460=121337,789553,329708
BC00461=121337,789553,329708
BC00462=167343,668969,639457
BC00463=382568,668969,422236
BC00464=299251,773200,237241
BC00465=299251,773200,237241
BC00466=299251,773200,237241
BC00467=299251,773200,237241
BC00468=299251,773200,237241
BC00469=299251,773200,237241
BC00470=279478,784302,237667
BC00471=279478,784302,237667
BC00472=279478,784302,237667
BC00473=279478,784302,237667
BC00474=279478,784302,237667
BC00475=279478,784302,237667
BC00476=280278,760811,181687
BC00477=280278,760811,181687
BC00478=280278,760811,181687
BC00479=280278,760811,181687
BC00480=280278,760811,181687
BC00481=280278,760811,181687
BC00482=277549,762343,181693
BC00483=277549,762343,181693
BC00484=277549,762343,181693
BC00485=277549,762343,181693
BC00486=277549,762343,181693
BC00487=277549,762343,181693
BC00488=297275,771567,184324
BC00489=335741,789553,189453
BC00490=335741,789553,189453
BC00491=335741,789553,189453
BC00492=335741,789553,189453
BC00493=335741,789553,189453
BC00494=335741,789553,189453
BC00495=351391,768330,121496
BC00496=351391,768330,121496
BC00497=351391,768330,121496
BC00498=351391,768330,121496
BC00499=351391,768330,121496
BC00500=351391,768330,121496
BC00501=283893,750061,250495
BC00502=283893,750061,250495
BC00503=165820,667836,534036
EC00000=798156,1112951
EC00001=798156,1112951
EC00002=798156,1112951
EC00003=798156,1112951
EC00004=798156,1112951
EC00005=798156,1112951
EC00006=798156,1112951
EC00007=798156,1112951
EC00008=798156,1112951
EC00009=798156,1112951
EC00010=798156,1112951
EC00011=798156,1112951
EC00012=798156,1112951
EC00013=798156,1112951
EC00014=798156,1112951
EC00015=798156,1112951
EC00016=798156,1112951
EC00017=798156,1112951
EC00018=798156,1112951
EC00019=798156,1112951
EC00020=798156,1112951
EC00021=798156,1112951
EC00022=798156,1112951
EC00023=798156,1112951
EC00024=798156,1112951
EC00025=798156,1112951
EC00026=798156,1112951
EC00027=798156,1112951
EC00028=798156,1112951
EC00029=798156,1112951
EC00030=798156,1112951
EC00031=798156,1112951
EC00032=798156,1112951
EC00033=798156,1112951
EC00034=798156,1112951
EC00035=798156,1112951
EC00036=798156,1112951
EC00037=798156,1112951
EC00038=798156,1112951
EC00039=798156,1112951
EC00040=798156,1112951
EC00041=798156,1112951
EC00042=798156,1112951
EC00043=798156,1112951
EC00044=798156,1112951
EC00045=798156,1112951
EC00046=798156,1112951
EC00047=798156,1112951
EC00048=798156,1112951
EC00049=798156,1112951
EC00050=798156,1112951
EC00051=798156,1112951
EC00052=798156,1112951
EC00053=798156,1112951
EC00054=798156,1112951
EC00055=798156,1112951
EC00056=798156,1112951
EC00057=798156,1112951
EC00058=798156,1112951
EC00059=798156,1112951
EC00060=798156,1112951
EC00061=798156,1112951
EC00062=798156,1112951
EC00063=798156,1112951
EC00064=798156,1112951
EC00065=798156,1112951
EC00066=798156,1112951
EC00067=798156,1112951
EC00068=798156,1112951
EC00069=798156,1112951
EC00070=798156,1112951
EC00071=798156,1112951
EC00072=798156,1112951
EC00073=798156,1112951
EC00074=798156,1112951
EC00075=798156,1112951
EC00076=798156,1112951
EC00077=798156,1112951
EC00078=798156,1112951
EC00079=798156,1112951
EC00080=798156,1112951
EC00081=798156,1112951
EC00082=798156,1112951
EC00083=798156,1112951
EC00084=798156,1112951
EC00085=798156,1112951
EC00086=798156,1112951
EC00087=798156,1112951
EC00088=798156,1112951
EC00089=798156,1112951
EC00090=798156,1112951
EC00091=798156,1112951
EC00092=798156,1112951
EC00093=798156,1112951
EC00094=798156,1112951
EC00095=798156,1112951
EC00096=798156,1112951
EC00097=798156,1112951
EC00098=798156,1112951
EC00099=798156,1112951
EC00100=798156,1112951
EC00101=798156,1112951
EC00102=798156,1112951
EC00103=798156,1112951
EC00104=798156,1112951
EC00105=798156,1112951
EC00106=798156,1112951
EC00107=798156,1112951
EC00108=798156,1112951
EC00109=798156,1112951
EC00110=798156,1112951
EC00111=798156,1112951
EC00112=798156,1112951
EC00113=798156,1112951
EC00114=798156,1112951
EC00115=798156,1112951
EC00116=798156,1112951
EC00117=798156,1112951
EC00118=798156,1112951
EC00119=798156,1112951
EC00120=798156,1112951
EC00121=798156,1112951
EC00122=798156,1112951
EC00123=798156,1112951
EC00124=798156,1112951
EC00125=798156,1112951
EC00126=798156,1112951
EC00127=798156,1112951
EC00128=798156,1112951
EC00129=798156,1112951
EC00130=798156,1112951
EC00131=798156,1112951
EC00132=798156,1112951
EC00133=798156,1112951
EC00134=798156,1112951
EC00135=798156,1112951
EC00136=798156,1112951
EC00137=798156,1112951
EC00138=798156,1112951
EC00139=798156,1112951
EC00140=798156,1112951
EC00141=798156,1112951
EC00142=798156,1112951
EC00143=798156,1112951
EC00144=798156,1112951
EC00145=798156,1112951
EC00146=798156,1112951
EC00147=798156,1112951
EC00148=798156,1112951
EC00149=798156,1112951
EC00150=798156,1112951
EC00151=798156,1112951
EC00152=798156,1112951
EC00153=798156,1112951
EC00154=798156,1112951
EC00155=798156,1112951
EC00156=798156,1112951
EC00157=798156,1112951
EC00158=798156,1112951
EC00159=798156,1112951
EC00160=798156,1112951
EC00161=798156,1112951
EC00162=798156,1112951
EC00163=798156,1112951
EC00164=798156,1112951
EC00165=798156,1112951
EC00166=798156,1112951
EC00167=798156,1112951
EC00168=798156,1112951
EC00169=798156,1112951
EC00170=798156,1112951
EC00171=798156,1112951
EC00172=798156,1112951
EC00173=798156,1112951
EC00174=798155,1112950
EC00175=798156,1112951
EC00176=798156,1112951
EC00177=798156,1112951
EC00178=798156,1112951
EC00179=798156,1112951
EC00180=798156,1112951
EC00181=798156,1112951
EC00182=798156,1112951
EC00183=798156,1112951
EC00184=798156,1112951
EC00185=798156,1112951
EC00186=798156,1112951
EC00187=798156,1112951
EC00188=798156,1112951
EC00189=798156,1112951
EC00190=798156,1112951
EC00191=798156,1112951
EC00192=798156,1112951
EC00193=798156,1112951
EC00194=798156,1112951
EC00195=798156,1112951
EC00196=798156,1112951
EC00197=798156,1112951
EC00198=798156,1112951
EC00199=798156,1112951
EC00200=798156,1112951
EC00201=798156,1112951
EC00202=798156,1112951
EC00203=798156,1112951
EC00204=798156,1112951
EC00205=798156,1112951
EC00206=798156,1112951
EC00207=798156,1112951
EC00208=798156,1112951
EC00209=798156,1112951
EC00210=798156,1112951
EC00211=798156,1112951
EC00212=798156,1112951
EC00213=798156,1112951
EC00214=798156,1112951
EC00215=798156,1112951
EC00216=798156,1112951
EC00217=798156,1112951
EC00218=798156,1112951
EC00219=798156,1112951
EC00220=798156,1112951
EC00221=798156,1112951
EC00222=798156,1112951
EC00223=798156,1112951
EC00224=798155,1112950
EC00225=798156,1112951
EC00226=798156,1112951
EC00227=798156,1112951
EC00228=798156,1112951
EC00229=798156,1112951
EC00230=798156,1112951
EC00231=798156,1112951
EC00232=798156,1112951
EC00233=798156,1112951
EC00234=798156,1112951
EC00235=798156,1112951
EC00236=798156,1112951
EC00237=798156,1112951
EC00238=798156,1112951
EC00239=798156,1112951
EC00240=798156,1112951
EC00241=798156,1112951
EC00242=798156,1112951
EC00243=798156,1112951
EC00244=798156,1112951
EC00245=798156,1112951
EC00246=798156,1112951
EC00247=798156,1112951
EC00248=798156,1112951
EC00249=798156,1112951
EC00250=798156,1112951
EC00251=798156,1112951
EC00252=798156,1112951
EC00253=798156,1112951
EC00254=798156,1112951
EC00255=798156,1112951
EC00256=798156,1112951
EC00257=798156,1112951
EC00258=798156,1112951
EC00259=798156,1112951
EC00260=798156,1112951
EC00261=798156,1112951
EC00262=798156,1112951
EC00263=798156,1112951
EC00264=798156,1112951
EC00265=798156,1112951
EC00266=798156,1112951
EC00267=798156,1112951
EC00268=798156,1112951
EC00269=798156,1112951
EC00270=798156,1112951
EC00271=798156,1112951
EC00272=798156,1112951
EC00273=798156,1112951
EC00274=798156,1112951
EC00275=798156,1112951
EC00276=798156,1112951
EC00277=798156,1112951
EC00278=798156,1112951
EC00279=798156,1112951
EC00280=798156,1112951
EC00281=798156,1112951
EC00282=798156,1112951
EC00283=798156,1112951
EC00284=798156,1112951
EC00285=798156,1112951
EC00286=798156,1112951
EC00287=798156,1112951
EC00288=798156,1112951
EC00289=798156,1112951
EC00290=798156,1112951
EC00291=798156,1112951
EC00292=798156,1112951
EC00293=798156,1112951
EC00294=798156,1112951
EC00295=798156,1112951
EC00296=798156,1112951
EC00297=798156,1112951
EC00298=798156,1112951
EC00299=798156,1112951
EC00300=798156,1112951
EC00301=798156,1112951
EC00302=798156,1112951
EC00303=798156,1112951
EC00304=798156,1112951
EC00305=798156,1112951
EC00306=798156,1112951
EC00307=798156,1112951
EC00308=798156,1112951
EC00309=798156,1112951
EC00310=798156,1112951
EC00311=798156,1112951
EC00312=798156,1112951
EC00313=798156,1112951
EC00314=798156,1112951
EC00315=798156,1112951
EC00316=798156,1112951
EC00317=798156,1112951
EC00318=798156,1112951
EC00319=798156,1112951
EC00320=798156,1112951
EC00321=798156,1112951
EC00322=798156,1112951
EC00323=798156,1112951
EC00324=798156,1112951
EC00325=798156,1112951
EC00326=798156,1112951
EC00327=798156,1112951
EC00328=798156,1112951
EC00329=798156,1112951
EC00330=798156,1112951
EC00331=798156,1112951
EC00332=798156,1112951
EC00333=798156,1112951
EC00334=798156,1112951
EC00335=798156,1112951
EC00336=798156,1112951
EC00337=798156,1112951
EC00338=798156,1112951
EC00339=798156,1112951
EC00340=798156,1112951
EC00341=798156,1112951
EC00342=798156,1112951
EC00343=798156,1112951
EC00344=798156,1112951
EC00345=798156,1112951
EC00346=798156,1112951
EC00347=798156,1112951
EC00348=798156,1112951
EC00349=798156,1112951
EC00350=798156,1112951
EC00351=798155,1112950
EC00352=798155,1112950
EC00353=798155,1112950
EC00354=798155,1112950
EC00355=798155,1112950
EC00356=798155,1112950
EC00357=798155,1112950
EC00358=798155,1112950
EC00359=798155,1112950
EC00360=798155,1112950
EC00361=798155,1112950
EC00362=798155,1112950
EC00363=798155,1112950
EC00364=798156,1112951
EC00365=798156,1112951
EC00366=798156,1112951
EC00367=798156,1112951
EC00368=798156,1112951
EC00369=798156,1112951
EC00370=798156,1112951
EC00371=798156,1112951
EC00372=798156,1112951
EC00373=798156,1112951
EC00374=798156,1112951
EC00375=798156,1112951
EC00376=798156,1112951
EC00377=798156,1112951
EC00378=798156,1112951
EC00379=798155,1112950
EC00380=798155,1112950
EC00381=798155,1112950
EC00382=798155,1112950
EC00383=798155,1112950
EC00384=798155,1112950
EC00385=798155,1112950
EC00386=798155,1112950
EC00387=798154,1112949
EC00388=798154,1112949
EC00389=798154,1112949
EC00390=798154,1112949
EC00391=798156,1112951
EC00392=798156,1112951
EC00393=798156,1112951
EC00394=798156,1112951
EC00395=798156,1112951
EC00396=798156,1112951
EC00397=798156,1112951
EC00398=798156,1112951
EC00399=798156,1112951
EC00400=798156,1112951
EC00401=798156,1112951
EC00402=798156,1112951
EC00403=798156,1112951
EC00404=798156,1112951
EC00405=798156,1112951
EC00406=798156,1112951
EC00407=798156,1112951
EC00408=798156,1112951
EC00409=798156,1112951
EC00410=798156,1112951
EC00411=798156,1112951
EC00412=798156,1112951
EC00413=798156,1112951
EC00414=798156,1112951
EC00415=798156,1112951
EC00416=798156,1112951
EC00417=798156,1112951
EC00418=798156,1112951
EC00419=798156,1112951
EC00420=798156,1112951
EC00421=798156,1112951
EC00422=798156,1112951
EC00423=798156,1112951
EC00424=798156,1112951
EC00425=798156,1112951
EC00426=798156,1112951
EC00427=798156,1112951
EC00428=798156,1112951
EC00429=798156,1112951
EC00430=798156,1112951
EC00431=798156,1112951
EC00432=798156,1112951
EC00433=798156,1112951
EC00434=798156,1112951
EC00435=798156,1112951
EC00436=798156,1112951
EC00437=798156,1112951
EC00438=798156,1112951
EC00439=798156,1112951
EC00440=798156,1112951
EC00441=798156,1112951
EC00442=798156,1112951
EC00443=798156,1112951
EC00444=798156,1112951
EC00445=798156,1112951
EC00446=798156,1112951
EC00447=798156,1112951
EC00448=798156,1112951
EC00449=798156,1112951
EC00450=798156,1112951
EC00451=798156,1112951
EC00452=798156,1112951
EC00453=798156,1112951
EC00454=798156,1112951
EC00455=798156,1112951
EC00456=798156,1112951
EC00457=798156,1112951
EC00458=798156,1112951
EC00459=798156,1112951
EC00460=798156,1112951
EC00461=798156,1112951
EC00462=798156,1112951
EC00463=798156,1112951
EC00464=798156,1112951
EC00465=798156,1112951
EC00466=798156,1112951
EC00467=798156,1112951
EC00468=798156,1112951
EC00469=798156,1112951
EC00470=798156,1112951
EC00471=798156,1112951
EC00472=798156,1112951
EC00473=798156,1112951
EC00474=798156,1112951
EC00475=798156,1112951
EC00476=798156,1112951
EC00477=798156,1112951
EC00478=798156,1112951
EC00479=798156,1112951
EC00480=798156,1112951
EC00481=798156,1112951
EC00482=798156,1112951
EC00483=798156,1112951
EC00484=798156,1112951
EC00485=798156,1112951
EC00486=798156,1112951
EC00487=798156,1112951
EC00488=798156,1112951
EC00489=798156,1112951
EC00490=798156,1112951
EC00491=798156,1112951
EC00492=798156,1112951
EC00493=798156,1112951
EC00494=798156,1112951
EC00495=798156,1112951
EC00496=798156,1112951
EC00497=798156,1112951
EC00498=798156,1112951
EC00499=798156,1112951
EC00500=798156,1112951
EC00501=798156,1112951
EC00502=798156,1112951
EC00503=798156,1112951
///POSTYPE BASE
///RECTAN
///RCONF 0,0,0,0,0,0,0,0,0,0,0,0,0,0,0,0,0,0,0,0,0,0,0,0
P00006=0.222,-3.123,-1.508,0.0000,0.0000,0.0000
P00021=-0.225,-6.128,-0.405,0.0000,0.0000,0.0000
P00022=0.222,-3.123,-1.508,0.0000,0.0000,0.0000
P00023=0.143,-0.036,0.682,0.0000,0.0000,0.0000
P00024=0.145,-0.552,1.326,0.0000,0.0000,0.0000
P00025=-2.003,0.006,0.728,0.0000,0.0000,0.0000
P00026=0.562,-0.002,-0.337,0.0000,0.0000,0.0000
P00027=-0.746,0.015,-9.096,0.0000,0.0000,0.0000
P00028=-2.237,-0.018,-7.702,0.0000,0.0000,0.0000
P00029=-2.156,-0.086,-4.681,0.0000,0.0000,0.0000
P00030=5.926,-4.294,-1.390,0.0000,0.0000,0.0000
P00031=1.853,-0.001,-1.549,0.0000,0.0000,0.0000
P00032=1.957,0.503,-7.217,0.0000,0.0000,0.0000
///RCONF 0,0,0,0,1,0,0,0,0,0,0,0,0,0,0,0,0,0,0,0,0,0,0,0
P00033=-0.123,0.612,-5.012,0.0000,0.0000,0.0000
///RCONF 0,0,0,0,0,0,0,0,0,0,0,0,0,0,0,0,0,0,0,0,0,0,0,0
P00034=-0.304,0.773,-2.693,0.0000,0.0000,0.0000
P00042=-0.217,1.941,0.413,0.0000,0.0000,0.0000
P00043=-0.044,-1.937,1.197,0.0000,0.0000,0.0000
P00044=0.687,-2.322,1.156,0.0000,0.0000,0.0000
P00045=-0.068,-0.810,1.603,0.0000,0.0000,0.0000
P00046=0.799,0.043,1.292,0.0000,0.0000,0.0000
///RCONF 0,1,0,0,0,0,0,0,0,0,0,0,0,0,0,0,0,0,0,0,0,0,0,0
P00047=-0.011,1.737,-0.646,0.0000,0.0000,0.0000
///RCONF 0,0,0,0,0,0,0,0,0,0,0,0,0,0,0,0,0,0,0,0,0,0,0,0
P00048=2.411,0.025,-0.606,0.0000,0.0000,0.0000
P00049=3.413,-3.572,-1.618,0.0000,0.0000,0.0000
P00050=4.296,-4.501,-0.826,0.0000,0.0000,0.0000
P00051=0.367,3.892,0.009,0.0000,0.0000,0.0000
P00052=0.088,2.832,-0.342,0.0000,0.0000,0.0000
P00053=0.134,6.594,0.107,0.0000,0.0000,0.0000
P00054=-0.103,6.509,-0.702,0.0000,0.0000,0.0000
P00055=-0.342,8.912,1.324,0.0000,0.0000,0.0000
P00060=2.327,-2.514,-2.692,0.0000,0.0000,0.0000
//INST
///DATE 2025/03/12 09:57
///ATTR SC,RW
///GROUP1 RB1,BS1
///GROUP2 ST1
NOP
'X2_38-47,64(1)(90,180)
'Down
MOVJ C00000 BC00000 VJ=100.00  +MOVJ EC00000 VJ=100.00
'Up
'Path S3659
SFTOF3D
MOVJ C00001 BC00001 VJ=100.00  +MOVJ EC00001 VJ=100.00
COMM PAUSE
COMM MOVL C00002 BC00002 V=666.7  +MOVJ EC00002 VJ=100.00
COMM SMOVL C00003 BC00003 V=166.7  +MOVJ EC00003
COMM SREFP 3 C00004 BC00004  +REFP EC00004
COMM CALL JOB:SEARCH-R1-S13D
COMM SET P021 P006
COMM SFTON3D P021
COMM SMOVL C00005 BC00005 V=166.7  +MOVJ EC00005
COMM SREFP 3 C00006 BC00006  +REFP EC00006
COMM CALL JOB:SEARCH-R1-S13D
COMM SET P021 P006
COMM SFTON3D P021
COMM SMOVL C00007 BC00007 V=166.7  +MOVJ EC00007
COMM MOVL C00008 BC00008 V=1000.0  +MOVJ EC00008 VJ=100.00
COMM 'EndPath S3659
COMM 'Path S4334
COMM SFTOF3D
COMM MOVJ C00009 BC00009 VJ=100.00  +MOVJ EC00009 VJ=100.00
COMM MOVL C00010 BC00010 V=666.7  +MOVJ EC00010 VJ=100.00
COMM SMOVL C00011 BC00011 V=166.7  +MOVJ EC00011
COMM SREFP 3 C00012 BC00012  +REFP EC00012
COMM CALL JOB:SEARCH-R1-S13D
COMM SET P022 P006
COMM SFTON3D P022
COMM SMOVL C00013 BC00013 V=166.7  +MOVJ EC00013
COMM SREFP 3 C00014 BC00014  +REFP EC00014
COMM CALL JOB:SEARCH-R1-S13D
COMM SET P022 P006
COMM SFTON3D P022
COMM SMOVL C00015 BC00015 V=166.7  +MOVJ EC00015
COMM MOVL C00016 BC00016 V=1000.0  +MOVJ EC00016 VJ=100.00
COMM 'EndPath S4334
COMM 'Path S3657
SFTOF3D
MOVJ C00017 BC00017 VJ=100.00  +MOVJ EC00017 VJ=100.00
MOVJ C00018 BC00018 VJ=100.00  +MOVJ EC00018 VJ=100.00
MOVL C00019 BC00019 V=666.7  +MOVJ EC00019 VJ=100.00
SMOVL C00020 BC00020 V=166.7  +MOVJ EC00020
SREFP 3 C00021 BC00021  +REFP EC00021
CALL JOB:SEARCH-R1-S13D
SET P023 P006
SFTON3D P023
SMOVL C00022 BC00022 V=166.7  +MOVJ EC00022
SREFP 3 C00023 BC00023  +REFP EC00023
CALL JOB:SEARCH-R1-S13D
SET P023 P006
SFTON3D P023
SMOVL C00024 BC00024 V=166.7  +MOVJ EC00024
SMOVL C00025 BC00025 V=500.0  +MOVJ EC00025
SMOVL C00026 BC00026 V=800.0  +MOVJ EC00026
SMOVL C00027 BC00027 V=166.7  +MOVJ EC00027
SREFP 3 C00028 BC00028  +REFP EC00028
CALL JOB:SEARCH-R1-S13D
SET P023 P006
SFTON3D P023
SMOVL C00029 BC00029 V=250.0  +MOVJ EC00029
MOVL C00030 BC00030 V=1000.0  +MOVJ EC00030 VJ=100.00
'EndPath S3657
MOVJ C00031 BC00031 VJ=100.00  +MOVJ EC00031 VJ=100.00
'Path S3665
SFTOF3D
MOVJ C00032 BC00032 VJ=100.00  +MOVJ EC00032 VJ=100.00
MOVL C00033 BC00033 V=800.0  +MOVJ EC00033 VJ=100.00
SMOVL C00034 BC00034 V=166.7  +MOVJ EC00034
SREFP 3 C00035 BC00035  +REFP EC00035
CALL JOB:SEARCH-R1-S13D
SET P024 P006
SFTON3D P024
SMOVL C00036 BC00036 V=166.7  +MOVJ EC00036
SMOVL C00037 BC00037 V=166.7  +MOVJ EC00037
SREFP 3 C00038 BC00038  +REFP EC00038
CALL JOB:SEARCH-R1-S13D
SET P024 P006
SFTON3D P024
SMOVL C00039 BC00039 V=166.7  +MOVJ EC00039
SMOVL C00040 BC00040 V=166.7  +MOVJ EC00040
SREFP 3 C00041 BC00041  +REFP EC00041
CALL JOB:SEARCH-R1-S13D
SET P024 P006
SFTON3D P024
SMOVL C00042 BC00042 V=166.7  +MOVJ EC00042
MOVL C00043 BC00043 V=1000.0  +MOVJ EC00043 VJ=100.00
MOVL C00044 BC00044 V=1000.0  +MOVJ EC00044 VJ=100.00
'EndPath S3665
'Path S4335
SFTOF3D
MOVJ C00045 BC00045 VJ=100.00  +MOVJ EC00045 VJ=100.00
MOVL C00046 BC00046 V=800.0  +MOVJ EC00046 VJ=100.00
SMOVL C00047 BC00047 V=166.7  +MOVJ EC00047
SREFP 3 C00048 BC00048  +REFP EC00048
CALL JOB:SEARCH-R1-S13D
SET P025 P006
SFTON3D P025
SMOVL C00049 BC00049 V=166.7  +MOVJ EC00049
SMOVL C00050 BC00050 V=166.7  +MOVJ EC00050
SREFP 3 C00051 BC00051  +REFP EC00051
CALL JOB:SEARCH-R1-S13D
SET P025 P006
SFTON3D P025
SMOVL C00052 BC00052 V=166.7  +MOVJ EC00052
SMOVL C00053 BC00053 V=166.7  +MOVJ EC00053
SREFP 3 C00054 BC00054  +REFP EC00054
CALL JOB:SEARCH-R1-S13D
SET P025 P006
SFTON3D P025
SMOVL C00055 BC00055 V=166.7  +MOVJ EC00055
MOVL C00056 BC00056 V=1000.0  +MOVJ EC00056 VJ=100.00
MOVL C00057 BC00057 V=1000.0  +MOVJ EC00057 VJ=100.00
'EndPath S4335
'Path S3666
SFTOF3D
MOVJ C00058 BC00058 VJ=100.00  +MOVJ EC00058 VJ=100.00
MOVL C00059 BC00059 V=800.0  +MOVJ EC00059 VJ=100.00
SMOVL C00060 BC00060 V=166.7  +MOVJ EC00060
SREFP 3 C00061 BC00061  +REFP EC00061
CALL JOB:SEARCH-R1-S13D
SET P026 P006
SFTON3D P026
SMOVL C00062 BC00062 V=166.7  +MOVJ EC00062
SREFP 3 C00063 BC00063  +REFP EC00063
CALL JOB:SEARCH-R1-S13D
SET P026 P006
SFTON3D P026
SMOVL C00064 BC00064 V=166.7  +MOVJ EC00064
MOVL C00065 BC00065 V=1000.0  +MOVJ EC00065 VJ=100.00
'EndPath S3666
MOVJ C00066 BC00066 VJ=100.00  +MOVJ EC00066 VJ=100.00
MOVJ C00067 BC00067 VJ=100.00  +MOVJ EC00067 VJ=100.00
'Path S3661
SFTOF3D
MOVJ C00068 BC00068 VJ=100.00  +MOVJ EC00068 VJ=100.00
MOVL C00069 BC00069 V=800.0  +MOVJ EC00069 VJ=100.00
SMOVL C00070 BC00070 V=166.7  +MOVJ EC00070
SREFP 3 C00071 BC00071  +REFP EC00071
CALL JOB:SEARCH-R1-S13D
SET P027 P006
SFTON3D P027
SMOVL C00072 BC00072 V=166.7  +MOVJ EC00072
SMOVL C00073 BC00073 V=166.7  +MOVJ EC00073
SREFP 3 C00074 BC00074  +REFP EC00074
CALL JOB:SEARCH-R1-S13D
SET P027 P006
SFTON3D P027
SMOVL C00075 BC00075 V=250.0  +MOVJ EC00075
SMOVL C00076 BC00076 V=166.7  +MOVJ EC00076
SREFP 3 C00077 BC00077  +REFP EC00077
CALL JOB:SEARCH-R1-S13D
SET P027 P006
SFTON3D P027
SMOVL C00078 BC00078 V=166.7  +MOVJ EC00078
MOVL C00079 BC00079 V=1000.0  +MOVJ EC00079 VJ=100.00
MOVL C00080 BC00080 V=1000.0  +MOVJ EC00080 VJ=100.00
'EndPath S3661
'Path S4336
SFTOF3D
MOVJ C00081 BC00081 VJ=100.00  +MOVJ EC00081 VJ=100.00
MOVL C00082 BC00082 V=800.0  +MOVJ EC00082 VJ=100.00
SMOVL C00083 BC00083 V=166.7  +MOVJ EC00083
SREFP 3 C00084 BC00084  +REFP EC00084
CALL JOB:SEARCH-R1-S13D
SET P028 P006
SFTON3D P028
SMOVL C00085 BC00085 V=166.7  +MOVJ EC00085
SREFP 3 C00086 BC00086  +REFP EC00086
CALL JOB:SEARCH-R1-S13D
SET P028 P006
SFTON3D P028
SMOVL C00087 BC00087 V=166.7  +MOVJ EC00087
MOVL C00088 BC00088 V=1000.0  +MOVJ EC00088 VJ=100.00
'EndPath S4336
MOVJ C00089 BC00089 VJ=100.00  +MOVJ EC00089 VJ=100.00
'Path S4879
SFTOF3D
MOVJ C00090 BC00090 VJ=100.00  +MOVJ EC00090 VJ=100.00
MOVL C00091 BC00091 V=800.0  +MOVJ EC00091 VJ=100.00
SMOVL C00092 BC00092 V=166.7  +MOVJ EC00092
SREFP 3 C00093 BC00093  +REFP EC00093
CALL JOB:SEARCH-R1-S13D
SET P060 P006
SFTON3D P060
SMOVL C00094 BC00094 V=166.7  +MOVJ EC00094
SMOVL C00095 BC00095 V=166.7  +MOVJ EC00095
SREFP 3 C00096 BC00096  +REFP EC00096
CALL JOB:SEARCH-R1-S13D
SET P060 P006
SFTON3D P060
SMOVL C00097 BC00097 V=166.7  +MOVJ EC00097
SMOVL C00098 BC00098 V=250.0  +MOVJ EC00098
SMOVL C00099 BC00099 V=166.7  +MOVJ EC00099
SREFP 3 C00100 BC00100  +REFP EC00100
CALL JOB:SEARCH-R1-S13D
SET P060 P006
SFTON3D P060
SMOVL C00101 BC00101 V=166.7  +MOVJ EC00101
MOVL C00102 BC00102 V=1000.0  +MOVJ EC00102 VJ=100.00
'EndPath S4879
MOVJ C00103 BC00103 VJ=100.00  +MOVJ EC00103 VJ=100.00
'Path S3664
SFTOF3D
COMM PAUSE
COMM MOVJ C00104 BC00104 VJ=100.00  +MOVJ EC00104 VJ=100.00
COMM MOVL C00105 BC00105 V=800.0  +MOVJ EC00105 VJ=100.00
COMM SMOVL C00106 BC00106 V=166.7  +MOVJ EC00106
COMM SREFP 3 C00107 BC00107  +REFP EC00107
COMM CALL JOB:SEARCH-R1-S13D
COMM SET P029 P006
COMM SFTON3D P029
COMM SMOVL C00108 BC00108 V=166.7  +MOVJ EC00108
COMM SREFP 3 C00109 BC00109  +REFP EC00109
COMM CALL JOB:SEARCH-R1-S13D
COMM SET P029 P006
COMM SFTON3D P029
COMM SMOVL C00110 BC00110 V=166.7  +MOVJ EC00110
COMM MOVL C00111 BC00111 V=1000.0  +MOVJ EC00111 VJ=100.00
COMM 'EndPath S3664
COMM 'Path S4337
COMM SFTOF3D
COMM MOVJ C00112 BC00112 VJ=100.00  +MOVJ EC00112 VJ=100.00
COMM MOVL C00113 BC00113 V=800.0  +MOVJ EC00113 VJ=100.00
COMM SMOVL C00114 BC00114 V=166.7  +MOVJ EC00114
COMM SREFP 3 C00115 BC00115  +REFP EC00115
COMM CALL JOB:SEARCH-R1-S13D
COMM SET P030 P006
COMM SFTON3D P030
COMM SMOVL C00116 BC00116 V=166.7  +MOVJ EC00116
COMM SREFP 3 C00117 BC00117  +REFP EC00117
COMM CALL JOB:SEARCH-R1-S13D
COMM SET P030 P006
COMM SFTON3D P030
COMM SMOVL C00118 BC00118 V=166.7  +MOVJ EC00118
COMM MOVL C00119 BC00119 V=800.0  +MOVJ EC00119 VJ=100.00
COMM MOVL C00120 BC00120 V=1000.0  +MOVJ EC00120 VJ=100.00
COMM 'EndPath S4337
MOVJ C00121 BC00121 VJ=100.00  +MOVJ EC00121 VJ=100.00
'Path S3663
SFTOF3D
MOVJ C00122 BC00122 VJ=100.00  +MOVJ EC00122 VJ=100.00
MOVL C00123 BC00123 V=800.0  +MOVJ EC00123 VJ=100.00
SMOVL C00124 BC00124 V=166.7  +MOVJ EC00124
SREFP 3 C00125 BC00125  +REFP EC00125
CALL JOB:SEARCH-R1-S13D
SET P031 P006
SFTON3D P031
SMOVL C00126 BC00126 V=166.7  +MOVJ EC00126
SREFP 3 C00127 BC00127  +REFP EC00127
CALL JOB:SEARCH-R1-S13D
SET P031 P006
SFTON3D P031
SMOVL C00128 BC00128 V=166.7  +MOVJ EC00128
SMOVL C00129 BC00129 V=166.7  +MOVJ EC00129
SREFP 3 C00130 BC00130  +REFP EC00130
CALL JOB:SEARCH-R1-S13D
SET P031 P006
SFTON3D P031
SMOVL C00131 BC00131 V=166.7  +MOVJ EC00131
MOVL C00132 BC00132 V=1000.0  +MOVJ EC00132 VJ=100.00
'EndPath S3663
MOVJ C00133 BC00133 VJ=100.00  +MOVJ EC00133 VJ=100.00
'Path S4338
SFTOF3D
MOVJ C00134 BC00134 VJ=100.00  +MOVJ EC00134 VJ=100.00
MOVL C00135 BC00135 V=800.0  +MOVJ EC00135 VJ=100.00
SMOVL C00136 BC00136 V=166.7  +MOVJ EC00136
SREFP 3 C00137 BC00137  +REFP EC00137
CALL JOB:SEARCH-R1-S13D
SET P032 P006
SFTON3D P032
SMOVL C00138 BC00138 V=166.7  +MOVJ EC00138
SREFP 3 C00139 BC00139  +REFP EC00139
CALL JOB:SEARCH-R1-S13D
SET P032 P006
SFTON3D P032
SMOVL C00140 BC00140 V=166.7  +MOVJ EC00140
SMOVL C00141 BC00141 V=166.7  +MOVJ EC00141
SREFP 3 C00142 BC00142  +REFP EC00142
CALL JOB:SEARCH-R1-S13D
SET P032 P006
SFTON3D P032
SMOVL C00143 BC00143 V=166.7  +MOVJ EC00143
MOVL C00144 BC00144 V=1000.0  +MOVJ EC00144 VJ=100.00
'EndPath S4338
MOVJ C00145 BC00145 VJ=100.00  +MOVJ EC00145 VJ=100.00
'Path S3662
SFTOF3D
MOVJ C00146 BC00146 VJ=100.00  +MOVJ EC00146 VJ=100.00
MOVL C00147 BC00147 V=800.0  +MOVJ EC00147 VJ=100.00
SMOVL C00148 BC00148 V=166.7  +MOVJ EC00148
SREFP 3 C00149 BC00149  +REFP EC00149
CALL JOB:SEARCH-R1-S13D
SET P033 P006
SFTON3D P033
SMOVL C00150 BC00150 V=166.7  +MOVJ EC00150
SREFP 3 C00151 BC00151  +REFP EC00151
CALL JOB:SEARCH-R1-S13D
SET P033 P006
SFTON3D P033
SMOVL C00152 BC00152 V=166.7  +MOVJ EC00152
MOVL C00153 BC00153 V=1000.0  +MOVJ EC00153 VJ=100.00
'EndPath S3662
'Path S4339
SFTOF3D
MOVJ C00154 BC00154 VJ=100.00  +MOVJ EC00154 VJ=100.00
MOVL C00155 BC00155 V=800.0  +MOVJ EC00155 VJ=100.00
SMOVL C00156 BC00156 V=166.7  +MOVJ EC00156
SREFP 3 C00157 BC00157  +REFP EC00157
CALL JOB:SEARCH-R1-S13D
SET P034 P006
SFTON3D P034
SMOVL C00158 BC00158 V=166.7  +MOVJ EC00158
SMOVL C00159 BC00159 V=166.7  +MOVJ EC00159
SREFP 3 C00160 BC00160  +REFP EC00160
CALL JOB:SEARCH-R1-S13D
SET P034 P006
SFTON3D P034
SMOVL C00161 BC00161 V=166.7  +MOVJ EC00161
SMOVL C00162 BC00162 V=166.7  +MOVJ EC00162
SREFP 3 C00163 BC00163  +REFP EC00163
CALL JOB:SEARCH-R1-S13D
SET P034 P006
SFTON3D P034
SMOVL C00164 BC00164 V=166.7  +MOVJ EC00164
MOVL C00165 BC00165 V=1000.0  +MOVJ EC00165 VJ=100.00
'EndPath S4339
MOVJ C00166 BC00166 VJ=100.00  +MOVJ EC00166 VJ=100.00
'Path W3667
SFTOF3D
SFTON3D P026
MOVJ C00167 BC00167 VJ=100.00  +MOVJ EC00167 VJ=100.00
SMOVL C00168 BC00168 V=800.0  +MOVJ EC00168
SREFP 1 C00169 BC00169  +REFP EC00169
SREFP 2 C00170 BC00170  +REFP EC00170
SMOVL C00171 BC00171 V=166.7 PL=0  +MOVJ EC00171
MACRO1 MJ#(0) ARGF21
ARCON
SWVON WEV#(100)
SMOVL C00172 BC00172 V=9.2  +MOVJ EC00172
SMOVL C00173 BC00173 V=9.2  +MOVJ EC00173
SMOVL C00174 BC00174 V=9.2  +MOVJ EC00174
ARCOF
SWVOF
SMOVL C00175 BC00175 V=800.0  +MOVJ EC00175
SMOVL C00176 BC00176 V=1000.0  +MOVJ EC00176
SFTOF3D
'EndPath W3667
MOVJ C00177 BC00177 VJ=100.00  +MOVJ EC00177 VJ=100.00
MOVJ C00178 BC00178 VJ=100.00  +MOVJ EC00178 VJ=100.00
'Path W3668
SSFTOF
SFTOF3D
SFTON3D P028
MOVJ C00179 BC00179 VJ=100.00  +MOVJ EC00179 VJ=100.00
SMOVL C00180 BC00180 V=800.0  +MOVJ EC00180
SREFP 1 C00181 BC00181  +REFP EC00181
SREFP 2 C00182 BC00182  +REFP EC00182
SMOVL C00183 BC00183 V=150.0 PL=0  +MOVJ EC00183
ARCON
SWVON WEV#(100)
SFTON3D P027
SMOVL C00184 BC00184 V=9.2  +MOVJ EC00184
SMOVL C00185 BC00185 V=9.2  +MOVJ EC00185
ARCOF
SWVOF
SMOVL C00186 BC00186 V=800.0  +MOVJ EC00186
SMOVL C00187 BC00187 V=1000.0  +MOVJ EC00187
SFTOF3D
'EndPath W3668
MOVJ C00188 BC00188 VJ=100.00  +MOVJ EC00188 VJ=100.00
COMM 'Path W4546
COMM PAUSE
COMM SFTOF3D
COMM SFTON3D P022
COMM MOVJ C00189 BC00189 VJ=100.00  +MOVJ EC00189 VJ=100.00
COMM SMOVL C00190 BC00190 V=800.0  +MOVJ EC00190
COMM SMOVL C00191 BC00191 V=150.0 PL=0  +MOVJ EC00191
COMM MACRO1 MJ#(0) ARGF9
COMM ARCON
COMM SWVON WEV#(10)
COMM SFTON3D P021
COMM SMOVL C00192 BC00192 V=10.0  +MOVJ EC00192
COMM ARCOF
COMM SWVOF
COMM SMOVL C00193 BC00193 V=800.0  +MOVJ EC00193
COMM SMOVL C00194 BC00194 V=1000.0  +MOVJ EC00194
COMM SFTOF3D
COMM 'EndPath W4546
COMM 'Path W4901
COMM SFTOF3D
SFTON3D P060
COMM MOVJ C00195 BC00195 VJ=100.00  +MOVJ EC00195 VJ=100.00
MOVJ C00196 BC00196 VJ=100.00  +MOVJ EC00196 VJ=100.00
MOVJ C00197 BC00197 VJ=100.00  +MOVJ EC00197 VJ=100.00
SMOVL C00198 BC00198 V=800.0  +MOVJ EC00198
SMOVL C00199 BC00199 V=150.0 PL=0  +MOVJ EC00199
MACRO1 MJ#(0) ARGF14
ARCON
SMOVL C00200 BC00200 V=10.8  +MOVJ EC00200
ARCOF
SMOVL C00201 BC00201 V=800.0  +MOVJ EC00201
SFTOF3D
'EndPath W4901
'Path W4880
SFTOF3D
SFTON3D P060
SMOVL C00202 BC00202 V=800.0  +MOVJ EC00202
SMOVL C00203 BC00203 V=150.0 PL=0  +MOVJ EC00203
ARCON
SMOVL C00204 BC00204 V=10.0  +MOVJ EC00204
SMOVL C00205 BC00205 V=10.0  +MOVJ EC00205
SMOVL C00206 BC00206 V=10.0  +MOVJ EC00206
ARCOF
SMOVL C00207 BC00207 V=800.0  +MOVJ EC00207
SMOVL C00208 BC00208 V=1000.0  +MOVJ EC00208
SFTOF3D
'EndPath W4880
MOVJ C00209 BC00209 VJ=100.00  +MOVJ EC00209 VJ=100.00
COMM PAUSE
COMM MOVJ C00210 BC00210 VJ=100.00  +MOVJ EC00210 VJ=100.00
COMM 'Path W4548
COMM SFTOF3D
COMM SFTON3D P030
COMM MOVJ C00211 BC00211 VJ=100.00  +MOVJ EC00211 VJ=100.00
COMM SMOVL C00212 BC00212 V=800.0  +MOVJ EC00212
COMM SMOVL C00213 BC00213 V=150.0 PL=0  +MOVJ EC00213
COMM MACRO1 MJ#(0) ARGF9
COMM ARCON
COMM SFTON3D P029
COMM SMOVL C00214 BC00214 V=10.0  +MOVJ EC00214
COMM SMOVL C00215 BC00215 V=10.0  +MOVJ EC00215
COMM ARCOF
COMM SMOVL C00216 BC00216 V=800.0  +MOVJ EC00216
COMM SMOVL C00217 BC00217 V=1000.0  +MOVJ EC00217
COMM SFTOF3D
COMM 'EndPath W4548
COMM MOVJ C00218 BC00218 VJ=100.00  +MOVJ EC00218 VJ=100.00
MOVJ C00219 BC00219 VJ=100.00  +MOVJ EC00219 VJ=100.00
'Path W3671
SFTOF3D
SFTON3D P033
MOVJ C00220 BC00220 VJ=100.00  +MOVJ EC00220 VJ=100.00
SMOVL C00221 BC00221 V=800.0  +MOVJ EC00221
SMOVL C00222 BC00222 V=166.7 PL=0  +MOVJ EC00222
MACRO1 MJ#(0) ARGF14
ARCON
SMOVL C00223 BC00223 V=9.2  +MOVJ EC00223
SFTON3D P034
SMOVL C00224 BC00224 V=9.2  +MOVJ EC00224
SMOVL C00225 BC00225 V=9.2  +MOVJ EC00225
ARCOF
SMOVL C00226 BC00226 V=800.0  +MOVJ EC00226
SMOVL C00227 BC00227 V=1000.0  +MOVJ EC00227
SFTOF3D
'EndPath W3671
MOVJ C00228 BC00228 VJ=100.00  +MOVJ EC00228 VJ=100.00
'Path W3672
SFTOF3D
SFTON3D P024
MOVJ C00229 BC00229 VJ=100.00  +MOVJ EC00229 VJ=100.00
SMOVL C00230 BC00230 V=800.0  +MOVJ EC00230
SMOVL C00231 BC00231 V=166.7 PL=0  +MOVJ EC00231
ARCON
SMOVL C00232 BC00232 V=9.2  +MOVJ EC00232
SFTON3D P025
SMOVL C00233 BC00233 V=9.2  +MOVJ EC00233
SMOVL C00234 BC00234 V=9.2  +MOVJ EC00234
ARCOF
SMOVL C00235 BC00235 V=800.0  +MOVJ EC00235
SMOVL C00236 BC00236 V=1000.0  +MOVJ EC00236
SFTOF3D
'EndPath W3672
MOVJ C00237 BC00237 VJ=100.00  +MOVJ EC00237 VJ=100.00
'Path W3673
SFTOF3D
SFTON3D P032
MOVJ C00238 BC00238 VJ=100.00  +MOVJ EC00238 VJ=100.00
SMOVL C00239 BC00239 V=800.0  +MOVJ EC00239
SMOVL C00240 BC00240 V=166.7 PL=0  +MOVJ EC00240
ARCON
SMOVL C00241 BC00241 V=9.2  +MOVJ EC00241
SFTON3D P031
SMOVL C00242 BC00242 V=9.2  +MOVJ EC00242
SMOVL C00243 BC00243 V=9.2  +MOVJ EC00243
ARCOF
SMOVL C00244 BC00244 V=800.0  +MOVJ EC00244
SMOVL C00245 BC00245 V=1000.0  +MOVJ EC00245
SFTOF3D
'EndPath W3673
MOVJ C00246 BC00246 VJ=100.00  +MOVJ EC00246 VJ=100.00
'
MOVJ C00247 BC00247 VJ=100.00  +MOVJ EC00247 VJ=100.00
JUMP *VV
MOVJ C00248 BC00248 VJ=100.00  +MOVJ EC00248 VJ=100.00
'Path W3680
SFTOF3D
SFTON3D P023
MOVJ C00249 BC00249 VJ=100.00  +MOVJ EC00249 VJ=100.00
SMOVL C00250 BC00250 V=800.0  +MOVJ EC00250
SMOVL C00251 BC00251 V=166.7 PL=0  +MOVJ EC00251
SMOVL C00252 BC00252 V=10.0  +MOVJ EC00252
SMOVL C00253 BC00253 V=33.3  +MOVJ EC00253
SMOVL C00254 BC00254 V=33.3  +MOVJ EC00254
SMOVL C00255 BC00255 V=33.3  +MOVJ EC00255
SMOVL C00256 BC00256 V=10.0  +MOVJ EC00256
SMOVL C00257 BC00257 V=10.0  +MOVJ EC00257
SMOVL C00258 BC00258 V=10.0  +MOVJ EC00258
SMOVL C00259 BC00259 V=10.0  +MOVJ EC00259
SMOVL C00260 BC00260 V=10.0  +MOVJ EC00260
ARCOF
SMOVL C00261 BC00261 V=800.0  +MOVJ EC00261
SMOVL C00262 BC00262 V=1000.0  +MOVJ EC00262
SFTOF3D
'EndPath W3680
'Path W3681
*VV
SFTOF3D
SFTON3D P023
MOVJ C00263 BC00263 VJ=100.00  +MOVJ EC00263 VJ=100.00
SMOVL C00264 BC00264 V=800.0  +MOVJ EC00264
MACRO1 MJ#(0) ARGF9
SMOVL C00265 BC00265 V=166.7 PL=0  +MOVJ EC00265
COMM SMOVL C00266 BC00266 V=150.0 PL=0  +MOVJ EC00266
COMM MACRO1 MJ#(0) ARGF9
COMM ARCON
COMM SMOVL C00267 BC00267 V=8.3  +MOVJ EC00267
COMM SMOVL C00268 BC00268 V=8.3  +MOVJ EC00268
COMM SMOVL C00269 BC00269 V=8.3  +MOVJ EC00269
ARCON
SMOVL C00270 BC00270 V=8.3  +MOVJ EC00270
SMOVL C00271 BC00271 V=8.3  +MOVJ EC00271
SMOVL C00272 BC00272 V=8.3  +MOVJ EC00272
SMOVL C00273 BC00273 V=8.3  +MOVJ EC00273
SMOVL C00274 BC00274 V=8.3  +MOVJ EC00274
SMOVL C00275 BC00275 V=8.3  +MOVJ EC00275
ARCOF
SMOVL C00276 BC00276 V=800.0  +MOVJ EC00276
SMOVL C00277 BC00277 V=1000.0  +MOVJ EC00277
SFTOF3D
'EndPath W3681
'Down
MOVJ C00278 BC00278 VJ=100.00  +MOVJ EC00278 VJ=100.00
CALL JOB:CLEAN-R1_KM_3P
'1
MOVJ C00279 BC00279 VJ=100.00  +MOVJ EC00279 VJ=100.00
MOVJ C00280 BC00280 VJ=100.00  +MOVJ EC00280 VJ=100.00
MOVJ C00281 BC00281 VJ=100.00  +MOVJ EC00281 VJ=100.00
'Path S4334
SFTOF3D
MOVJ C00282 BC00282 VJ=100.00  +MOVJ EC00282 VJ=100.00
MOVL C00283 BC00283 V=800.0  +MOVJ EC00283 VJ=100.00
SMOVL C00284 BC00284 V=166.7  +MOVJ EC00284
SREFP 3 C00285 BC00285  +REFP EC00285
CALL JOB:SEARCH-R1-S13D
SET P048 P006
SFTON3D P048
SMOVL C00286 BC00286 V=166.7  +MOVJ EC00286
SMOVL C00287 BC00287 V=166.7  +MOVJ EC00287
SREFP 3 C00288 BC00288  +REFP EC00288
CALL JOB:SEARCH-R1-S13D
SET P048 P006
SFTON3D P048
SMOVL C00289 BC00289 V=166.7  +MOVJ EC00289
MOVL C00290 BC00290 V=1000.0  +MOVJ EC00290 VJ=100.00
'EndPath S4334
'Path S4335
SFTOF3D
MOVJ C00291 BC00291 VJ=100.00  +MOVJ EC00291 VJ=100.00
MOVL C00292 BC00292 V=800.0  +MOVJ EC00292 VJ=100.00
SMOVL C00293 BC00293 V=166.7  +MOVJ EC00293
SREFP 3 C00294 BC00294  +REFP EC00294
CALL JOB:SEARCH-R1-S13D
SET P047 P006
SFTON3D P047
SMOVL C00295 BC00295 V=250.0  +MOVJ EC00295
SMOVL C00296 BC00296 V=166.7  +MOVJ EC00296
SREFP 3 C00297 BC00297  +REFP EC00297
CALL JOB:SEARCH-R1-S13D
SET P047 P006
SFTON3D P047
SMOVL C00298 BC00298 V=166.7  +MOVJ EC00298
MOVL C00299 BC00299 V=1000.0  +MOVJ EC00299 VJ=100.00
'EndPath S4335
MOVJ C00300 BC00300 VJ=100.00  +MOVJ EC00300 VJ=100.00
MOVJ C00301 BC00301 VJ=100.00  +MOVJ EC00301 VJ=100.00
MOVJ C00302 BC00302 VJ=100.00  +MOVJ EC00302 VJ=100.00
MOVJ C00303 BC00303 VJ=100.00  +MOVJ EC00303 VJ=100.00
'Path S4336
SFTOF3D
MOVJ C00304 BC00304 VJ=100.00  +MOVJ EC00304 VJ=100.00
MOVL C00305 BC00305 V=800.0  +MOVJ EC00305 VJ=100.00
SMOVL C00306 BC00306 V=166.7  +MOVJ EC00306
SREFP 3 C00307 BC00307  +REFP EC00307
CALL JOB:SEARCH-R1-S13D
SET P046 P006
SFTON3D P046
SMOVL C00308 BC00308 V=250.0  +MOVJ EC00308
SMOVL C00309 BC00309 V=166.7  +MOVJ EC00309
SREFP 3 C00310 BC00310  +REFP EC00310
CALL JOB:SEARCH-R1-S13D
SET P046 P006
SFTON3D P046
SMOVL C00311 BC00311 V=166.7  +MOVJ EC00311
MOVL C00312 BC00312 V=1000.0  +MOVJ EC00312 VJ=100.00
'EndPath S4336
'Path S4337
SFTOF3D
MOVJ C00313 BC00313 VJ=100.00  +MOVJ EC00313 VJ=100.00
MOVL C00314 BC00314 V=800.0  +MOVJ EC00314 VJ=100.00
SMOVL C00315 BC00315 V=166.7  +MOVJ EC00315
SREFP 3 C00316 BC00316  +REFP EC00316
CALL JOB:SEARCH-R1-S13D
SET P050 P006
SFTON3D P050
SMOVL C00317 BC00317 V=166.7  +MOVJ EC00317
SREFP 3 C00318 BC00318  +REFP EC00318
CALL JOB:SEARCH-R1-S13D
SET P050 P006
SFTON3D P050
SMOVL C00319 BC00319 V=166.7  +MOVJ EC00319
MOVL C00320 BC00320 V=1000.0  +MOVJ EC00320 VJ=100.00
'EndPath S4337
'Path S4338
SFTOF3D
MOVJ C00321 BC00321 VJ=100.00  +MOVJ EC00321 VJ=100.00
MOVL C00322 BC00322 V=666.7  +MOVJ EC00322 VJ=100.00
SMOVL C00323 BC00323 V=166.7  +MOVJ EC00323
SREFP 3 C00324 BC00324  +REFP EC00324
CALL JOB:SEARCH-R1-S13D
SET P051 P006
SFTON3D P051
SMOVL C00325 BC00325 V=166.7  +MOVJ EC00325
SREFP 3 C00326 BC00326  +REFP EC00326
CALL JOB:SEARCH-R1-S13D
SET P051 P006
SFTON3D P051
SMOVL C00327 BC00327 V=166.7  +MOVJ EC00327
SMOVL C00328 BC00328 V=166.7  +MOVJ EC00328
SMOVL C00329 BC00329 V=133.3  +MOVJ EC00329
SREFP 3 C00330 BC00330  +REFP EC00330
CALL JOB:SEARCH-R1-S13D
SET P051 P006
SFTON3D P051
SMOVL C00331 BC00331 V=250.0  +MOVJ EC00331
SMOVL C00332 BC00332 V=500.0  +MOVJ EC00332
'EndPath S4338
'Path S4339
SFTOF3D
MOVJ C00333 BC00333 VJ=100.00  +MOVJ EC00333 VJ=100.00
MOVL C00334 BC00334 V=800.0  +MOVJ EC00334 VJ=100.00
SMOVL C00335 BC00335 V=166.7  +MOVJ EC00335
SREFP 3 C00336 BC00336  +REFP EC00336
CALL JOB:SEARCH-R1-S13D
SET P055 P006
SFTON3D P055
SMOVL C00337 BC00337 V=166.7  +MOVJ EC00337
SMOVL C00338 BC00338 V=166.7  +MOVJ EC00338
SMOVL C00339 BC00339 V=166.7  +MOVJ EC00339
SREFP 3 C00340 BC00340  +REFP EC00340
CALL JOB:SEARCH-R1-S13D
SET P055 P006
SFTON3D P055
SMOVL C00341 BC00341 V=166.7  +MOVJ EC00341
SREFP 3 C00342 BC00342  +REFP EC00342
CALL JOB:SEARCH-R1-S13D
SET P045 P006
SFTON3D P045
SMOVL C00343 BC00343 V=166.7  +MOVJ EC00343
SMOVL C00344 BC00344 V=166.7  +MOVJ EC00344
SMOVL C00345 BC00345 V=166.7  +MOVJ EC00345
SREFP 3 C00346 BC00346  +REFP EC00346
CALL JOB:SEARCH-R1-S13D
SET P045 P006
SFTON3D P045
SMOVL C00347 BC00347 V=166.7  +MOVJ EC00347
MOVL C00348 BC00348 V=1000.0  +MOVJ EC00348 VJ=100.00
'EndPath S4142
'Path S4143
SFTOF3D
MOVJ C00349 BC00349 VJ=100.00  +MOVJ EC00349 VJ=100.00
MOVL C00350 BC00350 V=800.0  +MOVJ EC00350 VJ=100.00
SMOVL C00351 BC00351 V=166.7  +MOVJ EC00351
SREFP 3 C00352 BC00352  +REFP EC00352
CALL JOB:SEARCH-R1-S13D
SET P054 P006
SFTON3D P054
SMOVL C00353 BC00353 V=166.7  +MOVJ EC00353
SMOVL C00354 BC00354 V=166.7  +MOVJ EC00354
SMOVL C00355 BC00355 V=166.7  +MOVJ EC00355
SREFP 3 C00356 BC00356  +REFP EC00356
CALL JOB:SEARCH-R1-S13D
SET P054 P006
SFTON3D P054
SMOVL C00357 BC00357 V=166.7  +MOVJ EC00357
SREFP 3 C00358 BC00358  +REFP EC00358
CALL JOB:SEARCH-R1-S13D
SET P044 P006
SFTON3D P044
SMOVL C00359 BC00359 V=166.7  +MOVJ EC00359
SMOVL C00360 BC00360 V=166.7  +MOVJ EC00360
MOVL C00361 BC00361 V=166.7  +MOVJ EC00361 VJ=0.78
SREFP 3 C00362 BC00362  +REFP EC00362
CALL JOB:SEARCH-R1-S13D
SET P044 P006
SFTON3D P044
SMOVL C00363 BC00363 V=166.7  +MOVJ EC00363
MOVL C00364 BC00364 V=1000.0  +MOVJ EC00364 VJ=100.00
'Path S4341
SFTOF3D
MOVJ C00365 BC00365 VJ=100.00  +MOVJ EC00365 VJ=100.00
MOVL C00366 BC00366 V=800.0  +MOVJ EC00366 VJ=100.00
SMOVL C00367 BC00367 V=166.7  +MOVJ EC00367
SREFP 3 C00368 BC00368  +REFP EC00368
CALL JOB:SEARCH-R1-S13D
SET P049 P006
SFTON3D P049
SMOVL C00369 BC00369 V=166.7  +MOVJ EC00369
SMOVL C00370 BC00370 V=166.7  +MOVJ EC00370
SREFP 3 C00371 BC00371  +REFP EC00371
CALL JOB:SEARCH-R1-S13D
SET P049 P006
SFTON3D P049
SMOVL C00372 BC00372 V=166.7  +MOVJ EC00372
MOVL C00373 BC00373 V=1000.0  +MOVJ EC00373 VJ=100.00
'EndPath S4341
MOVJ C00374 BC00374 VJ=100.00  +MOVJ EC00374 VJ=100.00
MOVJ C00375 BC00375 VJ=100.00  +MOVJ EC00375 VJ=100.00
'Path S4342
SFTOF3D
MOVJ C00376 BC00376 VJ=100.00  +MOVJ EC00376 VJ=100.00
MOVL C00377 BC00377 V=800.0  +MOVJ EC00377 VJ=100.00
SMOVL C00378 BC00378 V=166.7  +MOVJ EC00378
SREFP 3 C00379 BC00379  +REFP EC00379
CALL JOB:SEARCH-R1-S13D
SET P053 P006
SFTON3D P053
SMOVL C00380 BC00380 V=166.7  +MOVJ EC00380
SMOVL C00381 BC00381 V=166.7  +MOVJ EC00381
MOVL C00382 BC00382 V=166.7  +MOVJ EC00382 VJ=0.78
SREFP 3 C00383 BC00383  +REFP EC00383
CALL JOB:SEARCH-R1-S13D
SET P053 P006
SFTON3D P053
SMOVL C00384 BC00384 V=166.7  +MOVJ EC00384
SREFP 3 C00385 BC00385  +REFP EC00385
CALL JOB:SEARCH-R1-S13D
SET P043 P006
SFTON3D P043
SMOVL C00386 BC00386 V=166.7  +MOVJ EC00386
SMOVL C00387 BC00387 V=166.7  +MOVJ EC00387
MOVL C00388 BC00388 V=166.7  +MOVJ EC00388 VJ=0.78
SREFP 3 C00389 BC00389  +REFP EC00389
CALL JOB:SEARCH-R1-S13D
SET P043 P006
SFTON3D P043
SMOVL C00390 BC00390 V=166.7  +MOVJ EC00390
MOVL C00391 BC00391 V=1000.0  +MOVJ EC00391 VJ=100.00
'EndPath S4144
'Path S4145
SFTOF3D
MOVJ C00392 BC00392 VJ=100.00  +MOVJ EC00392 VJ=100.00
MOVL C00393 BC00393 V=800.0  +MOVJ EC00393 VJ=100.00
SMOVL C00394 BC00394 V=166.7  +MOVJ EC00394
SREFP 3 C00395 BC00395  +REFP EC00395
CALL JOB:SEARCH-R1-S13D
SET P052 P006
SFTON3D P052
SMOVL C00396 BC00396 V=166.7  +MOVJ EC00396
SMOVL C00397 BC00397 V=166.7  +MOVJ EC00397
MOVL C00398 BC00398 V=166.7  +MOVJ EC00398 VJ=0.78
SREFP 3 C00399 BC00399  +REFP EC00399
CALL JOB:SEARCH-R1-S13D
SET P052 P006
SFTON3D P052
SMOVL C00400 BC00400 V=166.7  +MOVJ EC00400
SREFP 3 C00401 BC00401  +REFP EC00401
CALL JOB:SEARCH-R1-S13D
SET P042 P006
SFTON3D P042
SMOVL C00402 BC00402 V=166.7  +MOVJ EC00402
SMOVL C00403 BC00403 V=166.7  +MOVJ EC00403
MOVL C00404 BC00404 V=166.7  +MOVJ EC00404 VJ=0.78
SREFP 3 C00405 BC00405  +REFP EC00405
CALL JOB:SEARCH-R1-S13D
SET P042 P006
SFTON3D P042
SMOVL C00406 BC00406 V=166.7  +MOVJ EC00406
'EndPath S4343
MOVJ C00407 BC00407 VJ=100.00  +MOVJ EC00407 VJ=100.00
'
'Path W4344
SFTOF3D
SFTON3D P051
MOVJ C00408 BC00408 VJ=60.00  +MOVJ EC00408 VJ=20.00
SMOVL C00409 BC00409 V=500.0  +MOVJ EC00409
SMOVL C00410 BC00410 V=166.7 PL=0  +MOVJ EC00410
MACRO1 MJ#(0) ARGF14
ARCON
SMOVL C00411 BC00411 V=8.3  +MOVJ EC00411
ARCOF
SMOVL C00412 BC00412 V=800.0  +MOVJ EC00412
SMOVL C00413 BC00413 V=150.0  +MOVJ EC00413
ARCON
SMOVL C00414 BC00414 V=11.7  +MOVJ EC00414
ARCOF
SMOVL C00415 BC00415 V=250.0  +MOVJ EC00415
SMOVL C00416 BC00416 V=500.0  +MOVJ EC00416
SMOVL C00417 BC00417 V=1000.0  +MOVJ EC00417
SFTOF3D
'EndPath W4344
'Path W4345
SFTOF3D
SFTON3D P045
MOVJ C00418 BC00418 VJ=100.00  +MOVJ EC00418 VJ=100.00
SMOVL C00419 BC00419 V=800.0  +MOVJ EC00419
SMOVL C00420 BC00420 V=150.0 PL=0  +MOVJ EC00420
MACRO1 MJ#(0) ARGF21
ARCON
SMOVL C00421 BC00421 V=11.7  +MOVJ EC00421
ARCOF
SMOVL C00422 BC00422 V=800.0  +MOVJ EC00422
SMOVL C00423 BC00423 V=1000.0  +MOVJ EC00423
SFTOF3D
'EndPath W4345
'Path W4346
SFTOF3D
SFTON3D P045
MOVJ C00424 BC00424 VJ=100.00  +MOVJ EC00424 VJ=100.00
SMOVL C00425 BC00425 V=800.0  +MOVJ EC00425
SMOVL C00426 BC00426 V=150.0 PL=0  +MOVJ EC00426
ARCON
SMOVL C00427 BC00427 V=11.7  +MOVJ EC00427
ARCOF
SMOVL C00428 BC00428 V=800.0  +MOVJ EC00428
SMOVL C00429 BC00429 V=1000.0  +MOVJ EC00429
SFTOF3D
'EndPath W4346
'Path W4347
SFTOF3D
SFTON3D P049
MOVJ C00430 BC00430 VJ=100.00  +MOVJ EC00430 VJ=100.00
SMOVL C00431 BC00431 V=800.0  +MOVJ EC00431
SMOVL C00432 BC00432 V=150.0 PL=0  +MOVJ EC00432
ARCON
SMOVL C00433 BC00433 V=11.7  +MOVJ EC00433
ARCOF
SMOVL C00434 BC00434 V=800.0  +MOVJ EC00434
SMOVL C00435 BC00435 V=1000.0  +MOVJ EC00435
SFTOF3D
'EndPath W4347
'Path W4348
SFTOF3D
SFTON3D P050
MOVJ C00436 BC00436 VJ=100.00  +MOVJ EC00436 VJ=100.00
SMOVL C00437 BC00437 V=800.0  +MOVJ EC00437
SMOVL C00438 BC00438 V=150.0 PL=0  +MOVJ EC00438
ARCON
SMOVL C00439 BC00439 V=11.7  +MOVJ EC00439
ARCOF
SMOVL C00440 BC00440 V=800.0  +MOVJ EC00440
SMOVL C00441 BC00441 V=1000.0  +MOVJ EC00441
SFTOF3D
'EndPath W4348
MOVJ C00442 BC00442 VJ=100.00  +MOVJ EC00442 VJ=100.00
MOVJ C00443 BC00443 VJ=100.00  +MOVJ EC00443 VJ=100.00
'1
'uwaga na podajnik
'Path W4349
SFTOF3D
SFTON3D P048
MOVJ C00444 BC00444 VJ=100.00  +MOVJ EC00444 VJ=100.00
SMOVL C00445 BC00445 V=800.0  +MOVJ EC00445
SMOVL C00446 BC00446 V=150.0 PL=0  +MOVJ EC00446
ARCON
SMOVL C00447 BC00447 V=11.7  +MOVJ EC00447
ARCOF
SMOVL C00448 BC00448 V=800.0  +MOVJ EC00448
SMOVL C00449 BC00449 V=1000.0  +MOVJ EC00449
SFTOF3D
'EndPath W4349
'Path W4350
SFTOF3D
SFTON3D P048
MOVJ C00450 BC00450 VJ=100.00  +MOVJ EC00450 VJ=100.00
SMOVL C00451 BC00451 V=800.0  +MOVJ EC00451
SMOVL C00452 BC00452 V=150.0 PL=0  +MOVJ EC00452
ARCON
SMOVL C00453 BC00453 V=11.7  +MOVJ EC00453
ARCOF
SMOVL C00454 BC00454 V=800.0  +MOVJ EC00454
SMOVL C00455 BC00455 V=1000.0  +MOVJ EC00455
SFTOF3D
'EndPath W4350
'Path W4351
SFTOF3D
SFTON3D P047
MOVJ C00456 BC00456 VJ=100.00  +MOVJ EC00456 VJ=100.00
SMOVL C00457 BC00457 V=800.0  +MOVJ EC00457
SMOVL C00458 BC00458 V=150.0 PL=0  +MOVJ EC00458
ARCON
SMOVL C00459 BC00459 V=11.7  +MOVJ EC00459
ARCOF
SMOVL C00460 BC00460 V=800.0  +MOVJ EC00460
SMOVL C00461 BC00461 V=1000.0  +MOVJ EC00461
SFTOF3D
'EndPath W4351
'2
MOVJ C00462 BC00462 VJ=100.00  +MOVJ EC00462 VJ=100.00
MOVJ C00463 BC00463 VJ=100.00  +MOVJ EC00463 VJ=100.00
'Path W4352
SFTOF3D
SFTON3D P043
MOVJ C00464 BC00464 VJ=100.00  +MOVJ EC00464 VJ=100.00
SMOVL C00465 BC00465 V=800.0  +MOVJ EC00465
SMOVL C00466 BC00466 V=150.0 PL=0  +MOVJ EC00466
ARCON
SMOVL C00467 BC00467 V=11.7  +MOVJ EC00467
ARCOF
SMOVL C00468 BC00468 V=800.0  +MOVJ EC00468
SMOVL C00469 BC00469 V=1000.0  +MOVJ EC00469
SFTOF3D
'EndPath W4352
'Path W4353
SFTOF3D
SFTON3D P043
MOVJ C00470 BC00470 VJ=100.00  +MOVJ EC00470 VJ=100.00
SMOVL C00471 BC00471 V=800.0  +MOVJ EC00471
SMOVL C00472 BC00472 V=150.0 PL=0  +MOVJ EC00472
ARCON
SMOVL C00473 BC00473 V=11.7  +MOVJ EC00473
ARCOF
SMOVL C00474 BC00474 V=800.0  +MOVJ EC00474
SMOVL C00475 BC00475 V=1000.0  +MOVJ EC00475
SFTOF3D
'EndPath W4353
'Path W4354
SFTOF3D
SFTON3D P042
MOVJ C00476 BC00476 VJ=100.00  +MOVJ EC00476 VJ=100.00
SMOVL C00477 BC00477 V=800.0  +MOVJ EC00477
SMOVL C00478 BC00478 V=150.0 PL=0  +MOVJ EC00478
ARCON
SMOVL C00479 BC00479 V=11.7  +MOVJ EC00479
ARCOF
SMOVL C00480 BC00480 V=800.0  +MOVJ EC00480
SMOVL C00481 BC00481 V=1000.0  +MOVJ EC00481
SFTOF3D
'EndPath W4354
'Path W4355
SFTOF3D
SFTON3D P042
MOVJ C00482 BC00482 VJ=100.00  +MOVJ EC00482 VJ=100.00
SMOVL C00483 BC00483 V=800.0  +MOVJ EC00483
SMOVL C00484 BC00484 V=150.0 PL=0  +MOVJ EC00484
ARCON
SMOVL C00485 BC00485 V=11.7  +MOVJ EC00485
ARCOF
SMOVL C00486 BC00486 V=800.0  +MOVJ EC00486
SMOVL C00487 BC00487 V=1000.0  +MOVJ EC00487
SFTOF3D
'EndPath W4355
'3
MOVJ C00488 BC00488 VJ=100.00  +MOVJ EC00488 VJ=100.00
'Path W4356
SFTOF3D
SFTON3D P044
MOVJ C00489 BC00489 VJ=100.00  +MOVJ EC00489 VJ=100.00
SMOVL C00490 BC00490 V=800.0  +MOVJ EC00490
SMOVL C00491 BC00491 V=150.0 PL=0  +MOVJ EC00491
ARCON
SMOVL C00492 BC00492 V=11.7  +MOVJ EC00492
ARCOF
SMOVL C00493 BC00493 V=800.0  +MOVJ EC00493
SMOVL C00494 BC00494 V=1000.0  +MOVJ EC00494
SFTOF3D
'EndPath W4356
'Path W4357
SFTOF3D
SFTON3D P046
MOVJ C00495 BC00495 VJ=100.00  +MOVJ EC00495 VJ=100.00
SMOVL C00496 BC00496 V=800.0  +MOVJ EC00496
SMOVL C00497 BC00497 V=150.0 PL=0  +MOVJ EC00497
MACRO1 MJ#(0) ARGF14
ARCON
SMOVL C00498 BC00498 V=11.7  +MOVJ EC00498
ARCOF
SMOVL C00499 BC00499 V=800.0  +MOVJ EC00499
SMOVL C00500 BC00500 V=1000.0  +MOVJ EC00500
SFTOF3D
'EndPath W4357
MOVJ C00501 BC00501 VJ=100.00  +MOVJ EC00501 VJ=100.00
MOVJ C00502 BC00502 VJ=100.00  +MOVJ EC00502 VJ=100.00
MOVJ C00503 BC00503 VJ=100.00  +MOVJ EC00503 VJ=100.00
END
